KUKA KRL program: MyProgram_332().src

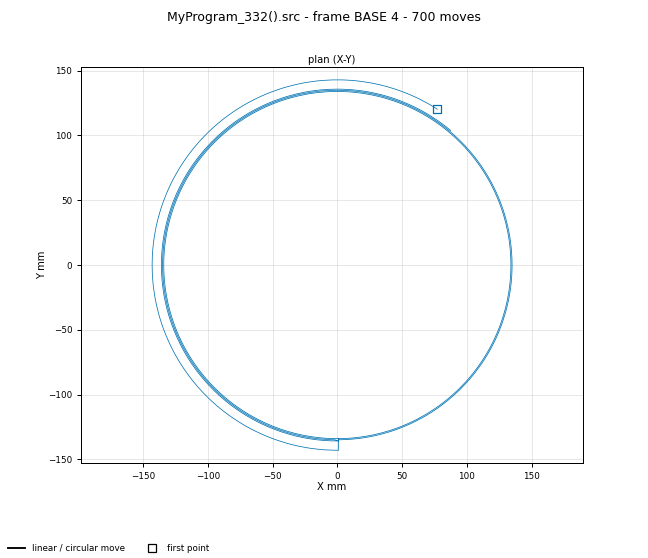
[picture p0: tool path of MyProgram_332().src in frame BASE 4, 700 of 700 moves have a stored position in this frame; points joined in program order, loops and branches not executed]
&ACCESS RVP
&REL 1
&PARAM TEMPLATE = C:\KRC\Roboter\Template\vorgabe
&PARAM EDITMASK = *
DEF MyProgram_332()
; ---- Setting reference (Base) ----
$BASE = BASE_DATA[4]

; --------------------------
; ---- Setting tool (TCP) ----
$TOOL = TOOL_DATA[3]
; --------------------------

$VEL.CP = VEL_APROX_PRINT
Startdeposition()
$VEL.CP = VEL_PRINT
LIN {X 77.191,Y 120.2651,Z 188,A 58.092,B 2.0692,C 0.0181,E1 2.1591,E2 395.982} C_DIS
LIN {X 74.024,Y 122.2399,Z 188,A 59.6872,B 2.0692,C 0.0151,E1 2.1552,E2 394.3743} C_DIS
LIN {X 70.243,Y 124.4513,Z 188,A 61.3886,B 2.0692,C 0.0127,E1 2.1511,E2 392.68} C_DIS
LIN {X 66.2155,Y 126.6377,Z 188,A 63.0311,B 2.0692,C 0.0112,E1 2.1471,E2 391.0624} C_DIS
LIN {X 63.4526,Y 128.0444,Z 188,A 64.253,B 2.0692,C 0.0096,E1 2.1441,E2 389.8433} C_DIS
LIN {X 60.2963,Y 129.5609,Z 188,A 65.6115,B 2.0692,C 0.008,E1 2.1406,E2 388.4907} C_DIS
LIN {X 55.8819,Y 131.5277,Z 188,A 67.6043,B 2.0692,C 0.0052,E1 2.1355,E2 386.4914} C_DIS
LIN {X 52.6403,Y 132.8581,Z 188,A 68.8611,B 2.0692,C 0.0043,E1 2.1323,E2 385.2535} C_DIS
LIN {X 48.7435,Y 134.3344,Z 188,A 70.5912,B 2.0692,C 0.0021,E1 2.1277,E2 383.5161} C_DIS
LIN {X 44.3687,Y 135.8443,Z 188,A 72.2898,B 2.0692,C 0.001,E1 2.1233,E2 381.8378} C_DIS
LIN {X 41.0274,Y 136.8906,Z 188,A 73.6584,B 2.0692,C -0.0002,E1 2.1196,E2 380.4739} C_DIS
LIN {X 37.6632,Y 137.8543,Z 188,A 75.0254,B 2.0692,C -0.0013,E1 2.116,E2 379.1118} C_DIS
LIN {X 34.5916,Y 138.6556,Z 188,A 76.3115,B 2.0692,C -0.0025,E1 2.1125,E2 377.8243} C_DIS
LIN {X 30.8569,Y 139.5349,Z 188,A 77.7931,B 2.0692,C -0.0035,E1 2.1084,E2 376.3503} C_DIS
LIN {X 27.4281,Y 140.2487,Z 188,A 79.1749,B 2.0692,C -0.0044,E1 2.1047,E2 374.9717} C_DIS
LIN {X 23.9731,Y 140.8799,Z 188,A 80.548,B 2.0692,C -0.0052,E1 2.1009,E2 373.6034} C_DIS
LIN {X 20.5127,Y 141.4248,Z 188,A 81.9382,B 2.0692,C -0.0059,E1 2.097,E2 372.2154} C_DIS
LIN {X 17.0406,Y 141.8848,Z 188,A 83.3239,B 2.0692,C -0.0066,E1 2.0932,E2 370.8325} C_DIS
LIN {X 13.9922,Y 142.2182,Z 188,A 84.541,B 2.0692,C -0.0072,E1 2.0898,E2 369.6174} C_DIS
LIN {X 10.0484,Y 142.5512,Z 188,A 86.0421,B 2.0692,C -0.0074,E1 2.0856,E2 368.1276} C_DIS
LIN {X 6.5517,Y 142.7556,Z 188,A 87.4775,B 2.0692,C -0.008,E1 2.0816,E2 366.6888} C_DIS
LIN {X 3.0497,Y 142.8736,Z 188,A 88.8217,B 2.0692,C -0.0081,E1 2.0779,E2 365.3528} C_DIS
LIN {X -0.4713,Y 142.9042,Z 188,A 90.1816,B 2.0692,C -0.0081,E1 2.0741,E2 363.9999} C_DIS
LIN {X -3.5202,Y 142.8619,Z 188,A 91.5285,B 2.0692,C -0.0089,E1 2.0703,E2 362.638} C_DIS
LIN {X -7.0204,Y 142.732,Z 188,A 92.9209,B 2.0692,C -0.009,E1 2.0664,E2 361.2477} C_DIS
LIN {X -10.515,Y 142.5171,Z 188,A 94.3659,B 2.0692,C -0.0092,E1 2.0623,E2 359.7981} C_DIS
LIN {X -14.0178,Y 142.2157,Z 188,A 95.7243,B 2.0692,C -0.0089,E1 2.0586,E2 358.4468} C_DIS
LIN {X -17.742,Y 141.8011,Z 188,A 97.2221,B 2.0692,C -0.0087,E1 2.0544,E2 356.9504} C_DIS
LIN {X -21.4322,Y 141.2887,Z 188,A 98.5946,B 2.0692,C -0.0079,E1 2.0506,E2 355.5936} C_DIS
LIN {X -24.4377,Y 140.8013,Z 188,A 99.9804,B 2.0692,C -0.0082,E1 2.0468,E2 354.1879} C_DIS
LIN {X -28.0983,Y 140.1152,Z 188,A 101.4739,B 2.0692,C -0.0077,E1 2.0427,E2 352.695} C_DIS
LIN {X -31.615,Y 139.3634,Z 188,A 102.9621,B 2.0692,C -0.0073,E1 2.0386,E2 351.2019} C_DIS
LIN {X -35.1507,Y 138.5137,Z 188,A 104.3003,B 2.0692,C -0.0061,E1 2.035,E2 349.8794} C_DIS
LIN {X -38.0927,Y 137.7342,Z 188,A 105.6465,B 2.0692,C -0.006,E1 2.0313,E2 348.5182} C_DIS
LIN {X -41.5005,Y 136.7458,Z 188,A 107.0908,B 2.0692,C -0.0052,E1 2.0274,E2 347.0718} C_DIS
LIN {X -44.8396,Y 135.6875,Z 188,A 108.5183,B 2.0692,C -0.0043,E1 2.0236,E2 345.6422} C_DIS
LIN {X -48.5796,Y 134.3935,Z 188,A 110.0373,B 2.0692,C -0.0029,E1 2.0196,E2 344.1326} C_DIS
LIN {X -51.4333,Y 133.3279,Z 188,A 111.38,B 2.0692,C -0.0023,E1 2.0161,E2 342.7755} C_DIS
LIN {X -54.7039,Y 132.0197,Z 188,A 112.8223,B 2.0692,C -0.0012,E1 2.0123,E2 341.3303} C_DIS
LIN {X -58.5883,Y 130.342,Z 188,A 114.6032,B 2.0692,C 0.0002,E1 2.0077,E2 339.5398} C_DIS
LIN {X -62.7858,Y 128.3734,Z 188,A 116.4246,B 2.0692,C 0.0022,E1 2.0031,E2 337.7243} C_DIS
LIN {X -66.0001,Y 126.7508,Z 188,A 118.0003,B 2.0692,C 0.0034,E1 1.9992,E2 336.1329} C_DIS
LIN {X -69.6929,Y 124.7605,Z 188,A 119.815,B 2.0692,C 0.005,E1 1.9947,E2 334.3027} C_DIS
LIN {X -73.4806,Y 122.5678,Z 188,A 121.54,B 2.0692,C 0.0073,E1 1.9905,E2 332.5826} C_DIS
LIN {X -77.1982,Y 120.2605,Z 188,A 123.3495,B 2.0692,C 0.0095,E1 1.9862,E2 330.7672} C_DIS
LIN {X -80.8424,Y 117.8416,Z 188,A 125.2463,B 2.0692,C 0.0116,E1 1.9818,E2 328.8536} C_DIS
LIN {X -84.6161,Y 115.1618,Z 188,A 127.1705,B 2.0692,C 0.0142,E1 1.9774,E2 326.9219} C_DIS
LIN {X -88.4338,Y 112.257,Z 188,A 129.1398,B 2.0692,C 0.0171,E1 1.9731,E2 324.9481} C_DIS
LIN {X -92.0062,Y 109.3481,Z 188,A 131.0239,B 2.0692,C 0.0201,E1 1.969,E2 323.0606} C_DIS
LIN {X -95.3272,Y 106.4653,Z 188,A 132.9387,B 2.0692,C 0.0228,E1 1.9649,E2 321.1277} C_DIS
LIN {X -98.5443,Y 103.4949,Z 188,A 134.7156,B 2.0692,C 0.0259,E1 1.9613,E2 319.3494} C_DIS
LIN {X -101.669,Y 100.4276,Z 188,A 136.5545,B 2.0691,C 0.029,E1 1.9576,E2 317.5011} C_DIS
LIN {X -104.6976,Y 97.2654,Z 188,A 138.3926,B 2.0691,C 0.0322,E1 1.9541,E2 315.6537} C_DIS
LIN {X -107.4912,Y 94.1692,Z 188,A 140.2044,B 2.069,C 0.0352,E1 1.9507,E2 313.8253} C_DIS
LIN {X -110.3256,Y 90.8325,Z 188,A 142.0599,B 2.069,C 0.0386,E1 1.9474,E2 311.9582} C_DIS
LIN {X -113.1958,Y 87.2296,Z 188,A 143.9226,B 2.0689,C 0.0425,E1 1.9441,E2 310.0948} C_DIS
LIN {X -115.4534,Y 84.219,Z 188,A 145.6429,B 2.0689,C 0.0454,E1 1.9412,E2 308.3484} C_DIS
LIN {X -117.9768,Y 80.6453,Z 188,A 147.4532,B 2.0687,C 0.0492,E1 1.9383,E2 306.5321} C_DIS
LIN {X -120.265,Y 77.1912,Z 188,A 149.2357,B 2.0687,C 0.0527,E1 1.9356,E2 304.7352} C_DIS
LIN {X -122.6861,Y 73.282,Z 188,A 151.1891,B 2.0685,C 0.0568,E1 1.9328,E2 302.7689} C_DIS
LIN {X -125.0733,Y 69.1289,Z 188,A 153.1628,B 2.0684,C 0.0613,E1 1.93,E2 300.7897} C_DIS
LIN {X -127.0339,Y 65.4554,Z 188,A 154.8401,B 2.0683,C 0.0654,E1 1.9279,E2 299.1126} C_DIS
LIN {X -128.5394,Y 62.4493,Z 188,A 156.4673,B 2.0682,C 0.0682,E1 1.9258,E2 297.4501} C_DIS
LIN {X -130.2908,Y 58.7026,Z 188,A 158.1973,B 2.068,C 0.0723,E1 1.9238,E2 295.7119} C_DIS
LIN {X -132.0308,Y 54.6774,Z 188,A 160.0188,B 2.0679,C 0.0766,E1 1.9218,E2 293.8834} C_DIS
LIN {X -133.4949,Y 51.0035,Z 188,A 161.6693,B 2.0677,C 0.0806,E1 1.9201,E2 292.2255} C_DIS
LIN {X -134.5486,Y 48.1494,Z 188,A 163.0215,B 2.0677,C 0.0836,E1 1.9188,E2 290.8568} C_DIS
LIN {X -135.8334,Y 44.4014,Z 188,A 164.6773,B 2.0674,C 0.0877,E1 1.9173,E2 289.1933} C_DIS
LIN {X -136.8857,Y 41.0433,Z 188,A 166.1859,B 2.0673,C 0.0913,E1 1.9161,E2 287.673} C_DIS
LIN {X -137.8633,Y 37.6301,Z 188,A 167.6986,B 2.0671,C 0.0949,E1 1.9149,E2 286.1495} C_DIS
LIN {X -138.639,Y 34.6571,Z 188,A 169.091,B 2.067,C 0.098,E1 1.914,E2 284.7367} C_DIS
LIN {X -139.5401,Y 30.8326,Z 188,A 170.7279,B 2.0668,C 0.1022,E1 1.9129,E2 283.0928} C_DIS
LIN {X -140.2508,Y 27.417,Z 188,A 172.2387,B 2.0666,C 0.1058,E1 1.9121,E2 281.568} C_DIS
LIN {X -140.8821,Y 23.9599,Z 188,A 173.5765,B 2.0664,C 0.1098,E1 1.9115,E2 280.2406} C_DIS
LIN {X -141.4257,Y 20.5062,Z 188,A 175.2435,B 2.0662,C 0.1133,E1 1.9107,E2 278.5393} C_DIS
LIN {X -141.8873,Y 17.0199,Z 188,A 176.7542,B 2.066,C 0.117,E1 1.9102,E2 277.0161} C_DIS
LIN {X -142.218,Y 13.9942,Z 188,A 178.0706,B 2.0658,C 0.1203,E1 1.9098,E2 275.6878} C_DIS
LIN {X -142.5505,Y 10.0574,Z 188,A 179.869,B 2.0656,C 0.1244,E1 1.9094,E2 273.8617} C_DIS
LIN {X -142.7564,Y 6.5367,Z 188,A -178.7374,B 2.0653,C 0.1284,E1 1.9092,E2 272.4718} C_DIS
LIN {X -142.8738,Y 3.0367,Z 188,A -177.1408,B 2.0651,C 0.132,E1 1.9092,E2 270.8502} C_DIS
LIN {X -142.9079,Y -0.008,Z 188,A -175.833,B 2.0649,C 0.1353,E1 1.9092,E2 269.5315} C_DIS
LIN {X -142.8622,Y -3.5089,Z 188,A -174.3736,B 2.0646,C 0.1391,E1 1.9092,E2 268.0654} C_DIS
LIN {X -142.7304,Y -7.0533,Z 188,A -172.8568,B 2.0644,C 0.1429,E1 1.9094,E2 266.5366} C_DIS
LIN {X -142.515,Y -10.5447,Z 188,A -171.3087,B 2.0641,C 0.1466,E1 1.9097,E2 264.9696} C_DIS
LIN {X -142.2149,Y -14.026,Z 188,A -169.8577,B 2.0638,C 0.1504,E1 1.9101,E2 263.5126} C_DIS
LIN {X -141.829,Y -17.5087,Z 188,A -168.3528,B 2.0636,C 0.1541,E1 1.9106,E2 261.9949} C_DIS
LIN {X -141.2849,Y -21.4566,Z 188,A -166.7811,B 2.0632,C 0.1586,E1 1.9112,E2 260.4277} C_DIS
LIN {X -140.7997,Y -24.4466,Z 188,A -165.3118,B 2.063,C 0.1615,E1 1.9119,E2 258.9244} C_DIS
LIN {X -140.1632,Y -27.8624,Z 188,A -163.7546,B 2.0627,C 0.165,E1 1.9127,E2 257.3455} C_DIS
LIN {X -139.4338,Y -31.307,Z 188,A -162.2535,B 2.0624,C 0.1687,E1 1.9136,E2 255.8329} C_DIS
LIN {X -138.5086,Y -35.1708,Z 188,A -160.7176,B 2.062,C 0.1731,E1 1.9146,E2 254.3056} C_DIS
LIN {X -137.7274,Y -38.1169,Z 188,A -159.2967,B 2.0618,C 0.176,E1 1.9157,E2 252.8579} C_DIS
LIN {X -136.7515,Y -41.482,Z 188,A -157.7941,B 2.0615,C 0.1796,E1 1.9169,E2 251.3426} C_DIS
LIN {X -135.6907,Y -44.8301,Z 188,A -156.2473,B 2.0612,C 0.183,E1 1.9182,E2 249.7774} C_DIS
LIN {X -134.3907,Y -48.5874,Z 188,A -154.503,B 2.0608,C 0.1869,E1 1.9199,E2 248.013} C_DIS
LIN {X -132.6867,Y -53.0655,Z 188,A -152.4738,B 2.0604,C 0.1916,E1 1.922,E2 245.9696} C_DIS
LIN {X -131.3491,Y -56.2955,Z 188,A -150.9828,B 2.0601,C 0.1949,E1 1.9236,E2 244.4668} C_DIS
LIN {X -129.9323,Y -59.4931,Z 188,A -149.5427,B 2.0598,C 0.1984,E1 1.9253,E2 243.0219} C_DIS
LIN {X -128.426,Y -62.6791,Z 188,A -148.0459,B 2.0594,C 0.2017,E1 1.9271,E2 241.5141} C_DIS
LIN {X -126.7358,Y -66.0287,Z 188,A -146.4049,B 2.0591,C 0.205,E1 1.9292,E2 239.8545} C_DIS
LIN {X -124.7679,Y -69.6797,Z 188,A -144.5415,B 2.0588,C 0.2086,E1 1.9317,E2 237.9637} C_DIS
LIN {X -122.575,Y -73.4685,Z 188,A -142.7546,B 2.0584,C 0.2126,E1 1.9343,E2 236.1729} C_DIS
LIN {X -120.2459,Y -77.221,Z 188,A -140.9018,B 2.058,C 0.2165,E1 1.9371,E2 234.3091} C_DIS
LIN {X -117.8382,Y -80.8473,Z 188,A -138.9752,B 2.0576,C 0.2199,E1 1.9401,E2 232.3575} C_DIS
LIN {X -115.1519,Y -84.6296,Z 188,A -137.0086,B 2.0572,C 0.2237,E1 1.9434,E2 230.3764} C_DIS
LIN {X -112.2516,Y -88.4406,Z 188,A -135.0163,B 2.0568,C 0.2276,E1 1.9468,E2 228.3743} C_DIS
LIN {X -109.3488,Y -92.0054,Z 188,A -133.1154,B 2.0563,C 0.2312,E1 1.9502,E2 226.4656} C_DIS
LIN {X -106.4681,Y -95.324,Z 188,A -131.193,B 2.056,C 0.2342,E1 1.9538,E2 224.5208} C_DIS
LIN {X -103.4984,Y -98.5407,Z 188,A -129.4109,B 2.0556,C 0.2375,E1 1.9572,E2 222.7351} C_DIS
LIN {X -100.4313,Y -101.6653,Z 188,A -127.5694,B 2.0553,C 0.2405,E1 1.9609,E2 220.8816} C_DIS
LIN {X -97.2556,Y -104.7068,Z 188,A -125.7391,B 2.0549,C 0.2435,E1 1.9646,E2 219.042} C_DIS
LIN {X -94.1794,Y -107.4823,Z 188,A -123.9498,B 2.0546,C 0.2459,E1 1.9684,E2 217.2346} C_DIS
LIN {X -90.8327,Y -110.3255,Z 188,A -122.1095,B 2.0543,C 0.2486,E1 1.9724,E2 215.3829} C_DIS
LIN {X -87.2268,Y -113.1979,Z 188,A -120.1487,B 2.054,C 0.2511,E1 1.9767,E2 213.4062} C_DIS
LIN {X -83.5252,Y -115.9562,Z 188,A -118.2289,B 2.0537,C 0.2536,E1 1.9811,E2 211.4764} C_DIS
LIN {X -80.1185,Y -118.3349,Z 188,A -116.5271,B 2.0534,C 0.2558,E1 1.985,E2 209.7695} C_DIS
LIN {X -76.4552,Y -120.7343,Z 188,A -114.7741,B 2.0531,C 0.2582,E1 1.9891,E2 208.0167} C_DIS
LIN {X -72.7203,Y -123.0205,Z 188,A -112.9568,B 2.0529,C 0.2602,E1 1.9935,E2 206.1906} C_DIS
LIN {X -68.8933,Y -125.2038,Z 188,A -111.1836,B 2.0526,C 0.2622,E1 1.9979,E2 204.4161} C_DIS
LIN {X -65.6011,Y -126.9597,Z 188,A -109.6543,B 2.0524,C 0.2638,E1 2.0017,E2 202.8819} C_DIS
LIN {X -62.4691,Y -128.5296,Z 188,A -108.2013,B 2.0523,C 0.265,E1 2.0053,E2 201.4217} C_DIS
LIN {X -58.7094,Y -130.2878,Z 188,A -106.4164,B 2.0521,C 0.2662,E1 2.0099,E2 199.6191} C_DIS
LIN {X -54.6923,Y -132.0246,Z 188,A -104.6725,B 2.0519,C 0.2678,E1 2.0144,E2 197.8764} C_DIS
LIN {X -51.0039,Y -133.4948,Z 188,A -102.9249,B 2.0519,C 0.2684,E1 2.019,E2 196.1061} C_DIS
LIN {X -46.0363,Y -135.2883,Z 188,A -100.9306,B 2.0516,C 0.2704,E1 2.0242,E2 194.129} C_DIS
LIN {X -42.7082,Y -136.3755,Z 188,A -99.5065,B 2.0515,C 0.2712,E1 2.0281,E2 192.7017} C_DIS
LIN {X -39.3559,Y -137.3805,Z 188,A -98.0852,B 2.0514,C 0.2719,E1 2.0319,E2 191.2773} C_DIS
LIN {X -36.4217,Y -138.1855,Z 188,A -96.8427,B 2.0513,C 0.2724,E1 2.0353,E2 190.0311} C_DIS
LIN {X -32.5698,Y -139.1453,Z 188,A -95.2317,B 2.0513,C 0.273,E1 2.0396,E2 188.417} C_DIS
LIN {X -29.1419,Y -139.9029,Z 188,A -93.8108,B 2.0512,C 0.2735,E1 2.0435,E2 186.9936} C_DIS
LIN {X -25.7011,Y -140.5752,Z 188,A -92.3963,B 2.0512,C 0.2739,E1 2.0474,E2 185.5772} C_DIS
LIN {X -22.7005,Y -141.0922,Z 188,A -91.0483,B 2.0512,C 0.2735,E1 2.0512,E2 184.2106} C_DIS
LIN {X -18.7821,Y -141.6649,Z 188,A -89.5751,B 2.051,C 0.2743,E1 2.0553,E2 182.7531} C_DIS
LIN {X -15.2873,Y -142.0844,Z 188,A -88.2632,B 2.051,C 0.2749,E1 2.0589,E2 181.455} C_DIS
LIN {X -12.2533,Y -142.3783,Z 188,A -86.8704,B 2.051,C 0.2741,E1 2.0628,E2 180.037} C_DIS
LIN {X -8.7592,Y -142.6358,Z 188,A -85.4919,B 2.051,C 0.2741,E1 2.0667,E2 178.6617} C_DIS
LIN {X -4.8038,Y -142.8258,Z 188,A -83.9134,B 2.051,C 0.2741,E1 2.0711,E2 177.0838} C_DIS
LIN {X -1.7417,Y -142.8954,Z 188,A -82.6323,B 2.0512,C 0.2735,E1 2.0747,E2 175.7945} C_DIS
LIN {X 1.0451,Y -142.9001,Z 188,A -81.9408,B 2.0509,C 0.2755,E1 2.0765,E2 175.1638} C_DIS
Enddeposition()
LIN {X 0.9696,Y -133.9381,Z 189,A -81.2734,B 1.7006,C 0.247,E1 1.727,E2 174.2111} C_DIS
Startdeposition()
$VEL.CP = VEL_PRINT
LIN {X -1.6562,Y -133.9352,Z 189,A -82.7535,B 1.7004,C 0.2488,E1 1.7227,E2 175.7398} C_DIS
LIN {X -4.9327,Y -133.8536,Z 189,A -84.2094,B 1.7003,C 0.2493,E1 1.7186,E2 177.2035} C_DIS
LIN {X -8.9898,Y -133.6442,Z 189,A -85.8795,B 1.7003,C 0.2492,E1 1.714,E2 178.8655} C_DIS
LIN {X -12.2534,Y -133.3835,Z 189,A -87.2736,B 1.7003,C 0.2492,E1 1.7101,E2 180.2593} C_DIS
LIN {X -15.6691,Y -133.0245,Z 189,A -88.7363,B 1.7003,C 0.2492,E1 1.706,E2 181.7218} C_DIS
LIN {X -18.9216,Y -132.6008,Z 189,A -90.1407,B 1.7003,C 0.249,E1 1.7021,E2 183.1269} C_DIS
LIN {X -22.1631,Y -132.0976,Z 189,A -91.551,B 1.7003,C 0.2488,E1 1.6982,E2 184.5387} C_DIS
LIN {X -25.4054,Y -131.5127,Z 189,A -92.9674,B 1.7004,C 0.2484,E1 1.6943,E2 185.9566} C_DIS
LIN {X -28.6288,Y -130.8491,Z 189,A -94.3882,B 1.7004,C 0.248,E1 1.6904,E2 187.3796} C_DIS
LIN {X -31.8278,Y -130.1082,Z 189,A -95.8093,B 1.7005,C 0.2476,E1 1.6865,E2 188.8034} C_DIS
LIN {X -35.0075,Y -129.2891,Z 189,A -97.2218,B 1.7006,C 0.247,E1 1.6827,E2 190.2175} C_DIS
LIN {X -38.1643,Y -128.3928,Z 189,A -98.6609,B 1.7007,C 0.2464,E1 1.6788,E2 191.6617} C_DIS
LIN {X -41.8745,Y -127.2307,Z 189,A -100.4022,B 1.7008,C 0.2456,E1 1.6741,E2 193.4139} C_DIS
LIN {X -45.1417,Y -126.108,Z 189,A -101.8618,B 1.701,C 0.2446,E1 1.6702,E2 194.8714} C_DIS
LIN {X -48.912,Y -124.6944,Z 189,A -103.6411,B 1.7011,C 0.2435,E1 1.6656,E2 196.6588} C_DIS
LIN {X -51.948,Y -123.4602,Z 189,A -105.064,B 1.7013,C 0.2424,E1 1.6619,E2 198.0848} C_DIS
LIN {X -54.9538,Y -122.1518,Z 189,A -106.5236,B 1.7014,C 0.2413,E1 1.6581,E2 199.5522} C_DIS
LIN {X -58.7511,Y -120.3724,Z 189,A -108.3429,B 1.7017,C 0.2396,E1 1.6535,E2 201.3753} C_DIS
LIN {X -61.6882,Y -118.8944,Z 189,A -109.7765,B 1.7019,C 0.2383,E1 1.6499,E2 202.8127} C_DIS
LIN {X -65.265,Y -116.9704,Z 189,A -111.6349,B 1.7021,C 0.2367,E1 1.6453,E2 204.6874} C_DIS
LIN {X -68.2395,Y -115.2603,Z 189,A -113.1191,B 1.7023,C 0.235,E1 1.6417,E2 206.1741} C_DIS
LIN {X -71.6626,Y -113.1633,Z 189,A -114.9315,B 1.7026,C 0.233,E1 1.6374,E2 207.9992} C_DIS
LIN {X -75.1549,Y -110.8746,Z 189,A -116.7644,B 1.7029,C 0.2307,E1 1.6331,E2 209.8385} C_DIS
LIN {X -77.7315,Y -109.0838,Z 189,A -118.1997,B 1.7031,C 0.2291,E1 1.6297,E2 211.2861} C_DIS
LIN {X -80.513,Y -107.0473,Z 189,A -119.6835,B 1.7034,C 0.2269,E1 1.6264,E2 212.7711} C_DIS
LIN {X -83.3511,Y -104.8524,Z 189,A -121.3995,B 1.7037,C 0.225,E1 1.6226,E2 214.5111} C_DIS
LIN {X -86.5851,Y -102.1983,Z 189,A -123.2754,B 1.704,C 0.2223,E1 1.6185,E2 216.3983} C_DIS
LIN {X -89.7072,Y -99.4696,Z 189,A -125.1588,B 1.7044,C 0.2195,E1 1.6145,E2 218.2961} C_DIS
LIN {X -92.719,Y -96.6678,Z 189,A -126.9845,B 1.7048,C 0.2165,E1 1.6108,E2 220.1303} C_DIS
LIN {X -95.5597,Y -93.8604,Z 189,A -128.8114,B 1.7051,C 0.2136,E1 1.6072,E2 221.9726} C_DIS
LIN {X -98.393,Y -90.8864,Z 189,A -130.6917,B 1.7055,C 0.2105,E1 1.6035,E2 223.8688} C_DIS
LIN {X -101.1837,Y -87.7692,Z 189,A -132.5791,B 1.7059,C 0.2072,E1 1.6,E2 225.7687} C_DIS
LIN {X -103.7757,Y -84.6879,Z 189,A -134.4013,B 1.7063,C 0.2038,E1 1.5967,E2 227.6035} C_DIS
LIN {X -106.3702,Y -81.4052,Z 189,A -136.3037,B 1.7067,C 0.2003,E1 1.5934,E2 229.5203} C_DIS
LIN {X -108.5512,Y -78.4735,Z 189,A -137.9487,B 1.7071,C 0.197,E1 1.5907,E2 231.1756} C_DIS
LIN {X -110.9952,Y -74.9767,Z 189,A -139.9984,B 1.7075,C 0.1933,E1 1.5874,E2 233.2539} C_DIS
LIN {X -113.1673,Y -71.6563,Z 189,A -141.6742,B 1.708,C 0.1895,E1 1.5849,E2 234.9265} C_DIS
LIN {X -114.8894,Y -68.8619,Z 189,A -143.3374,B 1.7083,C 0.1866,E1 1.5824,E2 236.6228} C_DIS
LIN {X -116.9818,Y -65.2446,Z 189,A -145.112,B 1.7088,C 0.1823,E1 1.58,E2 238.3953} C_DIS
LIN {X -118.8071,Y -61.8544,Z 189,A -146.9061,B 1.7092,C 0.1786,E1 1.5776,E2 240.2077} C_DIS
LIN {X -120.372,Y -58.7518,Z 189,A -148.4868,B 1.7095,C 0.175,E1 1.5756,E2 241.8} C_DIS
LIN {X -121.999,Y -55.2954,Z 189,A -150.3655,B 1.7099,C 0.1712,E1 1.5734,E2 243.7094} C_DIS
LIN {X -123.7488,Y -51.257,Z 189,A -152.2921,B 1.7104,C 0.1665,E1 1.5712,E2 245.6409} C_DIS
LIN {X -124.9682,Y -48.2075,Z 189,A -153.8327,B 1.7107,C 0.1631,E1 1.5697,E2 247.1983} C_DIS
LIN {X -126.4045,Y -44.3061,Z 189,A -155.9166,B 1.7111,C 0.1587,E1 1.5677,E2 249.3201} C_DIS
LIN {X -127.9219,Y -39.7142,Z 189,A -158.0785,B 1.7116,C 0.1533,E1 1.5658,E2 251.493} C_DIS
LIN {X -129.0888,Y -35.7373,Z 189,A -159.9092,B 1.712,C 0.1487,E1 1.5644,E2 253.3301} C_DIS
LIN {X -129.9304,Y -32.5454,Z 189,A -161.4449,B 1.7123,C 0.145,E1 1.5633,E2 254.8808} C_DIS
LIN {X -130.6896,Y -29.3499,Z 189,A -162.9723,B 1.7126,C 0.1412,E1 1.5623,E2 256.423} C_DIS
LIN {X -131.3708,Y -26.1344,Z 189,A -164.5006,B 1.7129,C 0.1375,E1 1.5615,E2 257.9659} C_DIS
LIN {X -131.9747,Y -22.8945,Z 189,A -166.0329,B 1.7132,C 0.1337,E1 1.5607,E2 259.5129} C_DIS
LIN {X -132.4964,Y -19.6519,Z 189,A -167.5916,B 1.7135,C 0.1299,E1 1.56,E2 261.0901} C_DIS
LIN {X -132.9006,Y -16.7013,Z 189,A -169.0642,B 1.7138,C 0.1265,E1 1.5595,E2 262.5868} C_DIS
LIN {X -133.2991,Y -13.1322,Z 189,A -170.6537,B 1.7141,C 0.1223,E1 1.559,E2 264.182} C_DIS
LIN {X -133.5815,Y -9.8488,Z 189,A -172.1826,B 1.7144,C 0.1184,E1 1.5587,E2 265.725} C_DIS
LIN {X -133.7949,Y -6.3332,Z 189,A -173.9256,B 1.7146,C 0.1144,E1 1.5584,E2 267.4964} C_DIS
LIN {X -133.923,Y -2.3881,Z 189,A -175.6855,B 1.715,C 0.1097,E1 1.5583,E2 269.264} C_DIS
LIN {X -133.9355,Y 1.6379,Z 189,A -177.5708,B 1.7152,C 0.1049,E1 1.5583,E2 271.1685} C_DIS
LIN {X -133.8537,Y 4.9287,Z 189,A -179.24,B 1.7155,C 0.1011,E1 1.5584,E2 272.8688} C_DIS
LIN {X -133.6462,Y 8.9572,Z 189,A 179.02,B 1.7158,C 0.0963,E1 1.5587,E2 274.6096} C_DIS
LIN {X -133.3858,Y 12.2294,Z 189,A 177.481,B 1.716,C 0.0925,E1 1.5591,E2 276.1642} C_DIS
LIN {X -133.0265,Y 15.6524,Z 189,A 175.8452,B 1.7162,C 0.0885,E1 1.5596,E2 277.819} C_DIS
LIN {X -132.4956,Y 19.6574,Z 189,A 174.0125,B 1.7164,C 0.0837,E1 1.5603,E2 279.6633} C_DIS
LIN {X -132.029,Y 22.5747,Z 189,A 172.568,B 1.7166,C 0.0803,E1 1.561,E2 281.1289} C_DIS
LIN {X -131.3718,Y 26.1298,Z 189,A 170.7691,B 1.7168,C 0.0762,E1 1.562,E2 282.9572} C_DIS
LIN {X -130.5677,Y 29.8837,Z 189,A 169.0808,B 1.717,C 0.0718,E1 1.563,E2 284.6499} C_DIS
LIN {X -129.5151,Y 34.1601,Z 189,A 167.082,B 1.7172,C 0.0668,E1 1.5644,E2 286.6613} C_DIS
LIN {X -128.3868,Y 38.1848,Z 189,A 165.1561,B 1.7173,C 0.0621,E1 1.5659,E2 288.6026} C_DIS
LIN {X -127.4124,Y 41.3202,Z 189,A 163.6391,B 1.7175,C 0.0584,E1 1.5672,E2 290.1321} C_DIS
LIN {X -126.3617,Y 44.4295,Z 189,A 162.1029,B 1.7175,C 0.0548,E1 1.5686,E2 291.6831} C_DIS
LIN {X -125.2905,Y 47.3642,Z 189,A 160.6527,B 1.7177,C 0.0514,E1 1.57,E2 293.1459} C_DIS
LIN {X -124.0329,Y 50.5669,Z 189,A 158.8948,B 1.7177,C 0.0478,E1 1.5719,E2 294.9367} C_DIS
LIN {X -122.4561,Y 54.2733,Z 189,A 157.2487,B 1.7179,C 0.0434,E1 1.5737,E2 296.5725} C_DIS
LIN {X -121.391,Y 56.6155,Z 189,A 155.8582,B 1.7179,C 0.0409,E1 1.5753,E2 297.9966} C_DIS
LIN {X -119.638,Y 60.2327,Z 189,A 154.1549,B 1.7181,C 0.0366,E1 1.5774,E2 299.6967} C_DIS
LIN {X -118.1271,Y 63.1467,Z 189,A 152.6371,B 1.7181,C 0.0333,E1 1.5794,E2 301.227} C_DIS
LIN {X -116.5454,Y 66.021,Z 189,A 150.99,B 1.7181,C 0.0302,E1 1.5817,E2 302.9016} C_DIS
LIN {X -114.4229,Y 69.6345,Z 189,A 149.1856,B 1.7183,C 0.026,E1 1.5843,E2 304.7062} C_DIS
LIN {X -112.6816,Y 72.4178,Z 189,A 147.6792,B 1.7183,C 0.0229,E1 1.5866,E2 306.2235} C_DIS
LIN {X -110.4528,Y 75.7734,Z 189,A 145.7927,B 1.7183,C 0.0191,E1 1.5896,E2 308.1279} C_DIS
LIN {X -108.0209,Y 79.2018,Z 189,A 143.9138,B 1.7183,C 0.0153,E1 1.5926,E2 310.0149} C_DIS
LIN {X -106.0981,Y 81.7603,Z 189,A 142.3569,B 1.7184,C 0.0126,E1 1.5953,E2 311.5926} C_DIS
LIN {X -103.5442,Y 84.9712,Z 189,A 140.4601,B 1.7184,C 0.0091,E1 1.5987,E2 313.5046} C_DIS
LIN {X -100.63,Y 88.4036,Z 189,A 138.4163,B 1.7184,C 0.0054,E1 1.6024,E2 315.5607} C_DIS
LIN {X -97.8243,Y 91.4982,Z 189,A 136.5504,B 1.7184,C 0.002,E1 1.606,E2 317.4345} C_DIS
LIN {X -94.9779,Y 94.449,Z 189,A 134.7023,B 1.7184,C -0.0012,E1 1.6096,E2 319.2921} C_DIS
LIN {X -92.0796,Y 97.277,Z 189,A 132.8399,B 1.7184,C -0.0041,E1 1.6134,E2 321.1683} C_DIS
LIN {X -89.0574,Y 100.0518,Z 189,A 130.9759,B 1.7184,C -0.007,E1 1.6173,E2 323.0436} C_DIS
LIN {X -85.9529,Y 102.7305,Z 189,A 129.1513,B 1.7184,C -0.0098,E1 1.6212,E2 324.8751} C_DIS
LIN {X -82.7673,Y 105.3138,Z 189,A 127.312,B 1.7184,C -0.0125,E1 1.6252,E2 326.7228} C_DIS
LIN {X -79.1869,Y 108.0318,Z 189,A 125.3488,B 1.7184,C -0.0153,E1 1.6297,E2 328.6893} C_DIS
LIN {X -75.7755,Y 110.4514,Z 189,A 123.5087,B 1.7184,C -0.0178,E1 1.6339,E2 330.5341} C_DIS
LIN {X -73.0462,Y 112.2751,Z 189,A 122.0421,B 1.7184,C -0.0196,E1 1.6373,E2 332.007} C_DIS
LIN {X -70.2594,Y 114.0399,Z 189,A 120.5811,B 1.7184,C -0.0213,E1 1.6408,E2 333.4727} C_DIS
LIN {X -66.8106,Y 116.0943,Z 189,A 118.7683,B 1.7183,C -0.0232,E1 1.6452,E2 335.2952} C_DIS
LIN {X -63.8176,Y 117.7662,Z 189,A 117.0997,B 1.7183,C -0.0245,E1 1.6494,E2 336.9858} C_DIS
LIN {X -60.5474,Y 119.4778,Z 189,A 115.5923,B 1.7183,C -0.0264,E1 1.6531,E2 338.4841} C_DIS
LIN {X -56.5809,Y 121.407,Z 189,A 113.6559,B 1.7183,C -0.0281,E1 1.658,E2 340.425} C_DIS
LIN {X -53.4468,Y 122.8187,Z 189,A 112.1862,B 1.7182,C -0.0295,E1 1.6618,E2 341.8937} C_DIS
LIN {X -49.8945,Y 124.304,Z 189,A 110.4685,B 1.7182,C -0.0307,E1 1.6663,E2 343.6185} C_DIS
LIN {X -45.9814,Y 125.8053,Z 189,A 108.6602,B 1.7182,C -0.032,E1 1.671,E2 345.4275} C_DIS
LIN {X -42.7433,Y 126.9414,Z 189,A 107.2026,B 1.7182,C -0.0331,E1 1.6749,E2 346.8831} C_DIS
LIN {X -39.7443,Y 127.9126,Z 189,A 105.6478,B 1.7182,C -0.0333,E1 1.6791,E2 348.4603} C_DIS
LIN {X -35.7151,Y 129.0949,Z 189,A 103.9618,B 1.7182,C -0.0346,E1 1.6836,E2 350.133} C_DIS
LIN {X -32.5393,Y 129.932,Z 189,A 102.5385,B 1.7181,C -0.0352,E1 1.6875,E2 351.5576} C_DIS
LIN {X -29.3438,Y 130.691,Z 189,A 101.1188,B 1.7181,C -0.0357,E1 1.6913,E2 352.9783} C_DIS
LIN {X -26.1308,Y 131.3716,Z 189,A 99.715,B 1.7181,C -0.0362,E1 1.6952,E2 354.3813} C_DIS
LIN {X -22.8752,Y 131.9782,Z 189,A 98.2755,B 1.7181,C -0.0365,E1 1.6992,E2 355.8227} C_DIS
LIN {X -19.6371,Y 132.4985,Z 189,A 96.8448,B 1.7181,C -0.0366,E1 1.7031,E2 357.2558} C_DIS
LIN {X -15.6659,Y 133.0249,Z 189,A 95.1237,B 1.7181,C -0.0368,E1 1.7079,E2 358.9769} C_DIS
LIN {X -12.2308,Y 133.3857,Z 189,A 93.6752,B 1.7181,C -0.0369,E1 1.712,E2 360.4215} C_DIS
LIN {X -8.9401,Y 133.6473,Z 189,A 92.2857,B 1.7181,C -0.0369,E1 1.7158,E2 361.8079} C_DIS
LIN {X -5.24,Y 133.8416,Z 189,A 90.6265,B 1.7181,C -0.0365,E1 1.7205,E2 363.4747} C_DIS
LIN {X -1.6342,Y 133.9355,Z 189,A 89.1182,B 1.7181,C -0.0363,E1 1.7247,E2 364.9785} C_DIS
LIN {X 2.3879,Y 133.923,Z 189,A 87.4179,B 1.7181,C -0.0359,E1 1.7295,E2 366.6759} C_DIS
LIN {X 5.6982,Y 133.8237,Z 189,A 86.0287,B 1.7181,C -0.0355,E1 1.7334,E2 368.0615} C_DIS
LIN {X 8.976,Y 133.6451,Z 189,A 84.6261,B 1.7181,C -0.035,E1 1.7373,E2 369.4634} C_DIS
LIN {X 12.2428,Y 133.3845,Z 189,A 83.2451,B 1.7181,C -0.0344,E1 1.7411,E2 370.8415} C_DIS
LIN {X 15.6618,Y 133.0254,Z 189,A 81.8067,B 1.7181,C -0.0337,E1 1.7451,E2 372.2758} C_DIS
LIN {X 18.9157,Y 132.6016,Z 189,A 80.4317,B 1.7181,C -0.0329,E1 1.749,E2 373.6471} C_DIS
LIN {X 22.1703,Y 132.0964,Z 189,A 79.0533,B 1.7181,C -0.0321,E1 1.7528,E2 375.0216} C_DIS
LIN {X 25.407,Y 131.5124,Z 189,A 77.6782,B 1.7181,C -0.0312,E1 1.7565,E2 376.3927} C_DIS
LIN {X 28.6253,Y 130.8499,Z 189,A 76.3064,B 1.7181,C -0.0302,E1 1.7603,E2 377.7603} C_DIS
LIN {X 31.8244,Y 130.109,Z 189,A 74.7915,B 1.7182,C -0.0285,E1 1.7644,E2 379.2873} C_DIS
LIN {X 36.1055,Y 128.9858,Z 189,A 73.0251,B 1.7182,C -0.0272,E1 1.7692,E2 381.0389} C_DIS
LIN {X 39.7914,Y 127.8982,Z 189,A 71.4996,B 1.7182,C -0.026,E1 1.7732,E2 382.5507} C_DIS
LIN {X 42.7506,Y 126.939,Z 189,A 70.1696,B 1.7182,C -0.0246,E1 1.7768,E2 383.8802} C_DIS
LIN {X 46.6769,Y 125.5479,Z 189,A 68.3549,B 1.7183,C -0.0224,E1 1.7816,E2 385.6983} C_DIS
LIN {X 50.5719,Y 124.0309,Z 189,A 66.6187,B 1.7183,C -0.0204,E1 1.7861,E2 387.4283} C_DIS
LIN {X 54.959,Y 122.1494,Z 189,A 64.7783,B 1.7183,C -0.0187,E1 1.7907,E2 389.2455} C_DIS
LIN {X 57.9375,Y 120.765,Z 189,A 63.3815,B 1.7183,C -0.0167,E1 1.7943,E2 390.6412} C_DIS
LIN {X 61.0641,Y 119.2148,Z 189,A 61.9242,B 1.7183,C -0.0147,E1 1.7979,E2 392.0943} C_DIS
LIN {X 65.2607,Y 116.9728,Z 189,A 60.0374,B 1.7184,C -0.0124,E1 1.8025,E2 393.964} C_DIS
LIN {X 68.8656,Y 114.8872,Z 189,A 58.3506,B 1.7184,C -0.0101,E1 1.8066,E2 395.6398} C_DIS
LIN {X 72.4087,Y 112.6875,Z 189,A 56.6652,B 1.7184,C -0.0076,E1 1.8105,E2 397.3138} C_DIS
LIN {X 75.1637,Y 110.8686,Z 189,A 55.3267,B 1.7184,C -0.0056,E1 1.8136,E2 398.6438} C_DIS
LIN {X 78.3762,Y 108.6217,Z 189,A 53.7098,B 1.7184,C -0.0029,E1 1.8173,E2 400.2537} C_DIS
LIN {X 81.4086,Y 106.3676,Z 189,A 52.135,B 1.7184,C -0.0002,E1 1.8208,E2 401.8238} C_DIS
LIN {X 84.69,Y 103.774,Z 189,A 50.4436,B 1.7184,C 0.0027,E1 1.8245,E2 403.5038} C_DIS
LIN {X 87.7693,Y 101.1837,Z 189,A 48.7866,B 1.7184,C 0.0057,E1 1.828,E2 405.1535} C_DIS
LIN {X 90.8859,Y 98.3935,Z 189,A 47.1224,B 1.7184,C 0.0086,E1 1.8314,E2 406.8033} C_DIS
LIN {X 93.857,Y 95.563,Z 189,A 45.7049,B 1.7184,C 0.0102,E1 1.8342,E2 408.1815} C_DIS
LIN {X 95.8767,Y 93.5372,Z 189,A 44.3141,B 1.7184,C 0.0138,E1 1.837,E2 409.5921} C_DIS
LIN {X 98.6965,Y 90.5563,Z 189,A 42.6836,B 1.7184,C 0.0168,E1 1.84,E2 411.2082} C_DIS
LIN {X 101.4246,Y 87.4899,Z 189,A 41.0248,B 1.7184,C 0.0201,E1 1.8431,E2 412.8559} C_DIS
LIN {X 104.0576,Y 84.3418,Z 189,A 39.3684,B 1.7183,C 0.0235,E1 1.846,E2 414.501} C_DIS
LIN {X 106.5995,Y 81.1054,Z 189,A 37.6753,B 1.7183,C 0.0271,E1 1.8489,E2 416.1865} C_DIS
LIN {X 109.0846,Y 77.7305,Z 189,A 35.9807,B 1.7182,C 0.0308,E1 1.8516,E2 417.8699} C_DIS
LIN {X 111.3789,Y 74.4055,Z 189,A 34.3777,B 1.7182,C 0.0341,E1 1.8541,E2 419.4585} C_DIS
LIN {X 113.9349,Y 70.4302,Z 189,A 32.5814,B 1.718,C 0.0376,E1 1.8568,E2 421.2286} C_DIS
LIN {X 116.099,Y 66.8025,Z 189,A 30.9107,B 1.718,C 0.0412,E1 1.8591,E2 422.8837} C_DIS
LIN {X 117.7773,Y 63.7973,Z 189,A 29.4125,B 1.7179,C 0.0451,E1 1.8611,E2 424.3854} C_DIS
LIN {X 119.6413,Y 60.2262,Z 189,A 27.9554,B 1.7178,C 0.0478,E1 1.863,E2 425.8112} C_DIS
LIN {X 121.4063,Y 56.5823,Z 189,A 26.3168,B 1.7177,C 0.0516,E1 1.8649,E2 427.4391} C_DIS
LIN {X 123.1108,Y 52.7713,Z 189,A 24.6653,B 1.7176,C 0.0554,E1 1.8668,E2 429.0751} C_DIS
LIN {X 124.6964,Y 48.9068,Z 189,A 23.0378,B 1.7174,C 0.0591,E1 1.8684,E2 430.6841} C_DIS
LIN {X 126.0063,Y 45.4239,Z 189,A 21.5127,B 1.7174,C 0.0629,E1 1.8699,E2 432.2017} C_DIS
LIN {X 127.4141,Y 41.3148,Z 189,A 19.8361,B 1.7172,C 0.0666,E1 1.8714,E2 433.8572} C_DIS
LIN {X 128.5348,Y 37.6793,Z 189,A 18.2729,B 1.717,C 0.0706,E1 1.8726,E2 435.4133} C_DIS
LIN {X 129.5213,Y 34.1368,Z 189,A 16.8767,B 1.7169,C 0.0737,E1 1.8736,E2 436.7887} C_DIS
LIN {X 130.3195,Y 30.9513,Z 189,A 15.5782,B 1.7167,C 0.0769,E1 1.8745,E2 438.0749} C_DIS
LIN {X 131.0396,Y 27.7466,Z 189,A 14.28,B 1.7166,C 0.08,E1 1.8753,E2 439.3607} C_DIS
LIN {X 131.6842,Y 24.5086,Z 189,A 12.9776,B 1.7164,C 0.0832,E1 1.8759,E2 440.6503} C_DIS
LIN {X 132.1857,Y 21.6356,Z 189,A 11.7812,B 1.7163,C 0.0863,E1 1.8765,E2 441.8411} C_DIS
LIN {X 132.7267,Y 18.0278,Z 189,A 10.2663,B 1.7161,C 0.0903,E1 1.8771,E2 443.3512} C_DIS
LIN {X 133.2279,Y 13.8411,Z 189,A 8.7181,B 1.7159,C 0.0936,E1 1.8776,E2 444.8689} C_DIS
LIN {X 133.5277,Y 10.5764,Z 189,A 7.4128,B 1.7157,C 0.0969,E1 1.8779,E2 446.1631} C_DIS
LIN {X 133.738,Y 7.4645,Z 189,A 6.2055,B 1.7156,C 0.0997,E1 1.8781,E2 447.3554} C_DIS
LIN {X 133.8794,Y 4.1901,Z 189,A 4.8367,B 1.7153,C 0.1034,E1 1.8782,E2 448.7208} C_DIS
LIN {X 133.9452,Y 0.4417,Z 189,A 3.3131,B 1.7151,C 0.1074,E1 1.8782,E2 450.2355} C_DIS
LIN {X 133.909,Y -3.1266,Z 189,A 1.9344,B 1.7149,C 0.1106,E1 1.8782,E2 451.5967} C_DIS
LIN {X 133.7372,Y -7.4799,Z 189,A 0.2912,B 1.7146,C 0.1144,E1 1.878,E2 453.2136} C_DIS
LIN {X 133.5264,Y -10.5915,Z 189,A -0.978,B 1.7144,C 0.1176,E1 1.8777,E2 454.4754} C_DIS
LIN {X 133.2232,Y -13.8843,Z 189,A -2.3138,B 1.7142,C 0.1211,E1 1.8774,E2 455.8022} C_DIS
LIN {X 132.8222,Y -17.2993,Z 189,A -3.6317,B 1.714,C 0.1241,E1 1.8769,E2 457.1019} C_DIS
LIN {X 132.3584,Y -20.5487,Z 189,A -4.9272,B 1.7137,C 0.1273,E1 1.8764,E2 458.3846} C_DIS
LIN {X 131.8151,Y -23.7861,Z 189,A -6.2241,B 1.7135,C 0.1304,E1 1.8758,E2 459.6689} C_DIS
LIN {X 131.1929,Y -27.0091,Z 189,A -7.5221,B 1.7133,C 0.1336,E1 1.8751,E2 460.9544} C_DIS
LIN {X 130.492,Y -30.2152,Z 189,A -8.8225,B 1.713,C 0.1367,E1 1.8743,E2 462.2428} C_DIS
LIN {X 129.7084,Y -33.4201,Z 189,A -10.128,B 1.7128,C 0.1398,E1 1.8734,E2 463.5358} C_DIS
LIN {X 128.8787,Y -36.4883,Z 189,A -11.3991,B 1.7125,C 0.1429,E1 1.8725,E2 464.7966} C_DIS
LIN {X 127.9024,Y -39.7777,Z 189,A -12.748,B 1.7122,C 0.1461,E1 1.8714,E2 466.1314} C_DIS
LIN {X 126.9431,Y -42.7382,Z 189,A -13.9946,B 1.712,C 0.1491,E1 1.8703,E2 467.3682} C_DIS
LIN {X 125.8065,Y -45.9781,Z 189,A -15.3369,B 1.7117,C 0.1522,E1 1.8691,E2 468.6954} C_DIS
LIN {X 124.7015,Y -48.8935,Z 189,A -16.5971,B 1.7114,C 0.1552,E1 1.8678,E2 469.9472} C_DIS
LIN {X 123.1152,Y -52.7609,Z 189,A -18.3813,B 1.711,C 0.1599,E1 1.8659,E2 471.7321} C_DIS
LIN {X 121.4015,Y -56.5927,Z 189,A -19.8974,B 1.7107,C 0.1626,E1 1.8642,E2 473.2137} C_DIS
LIN {X 119.8623,Y -59.7852,Z 189,A -21.3983,B 1.7104,C 0.1664,E1 1.8623,E2 474.7139} C_DIS
LIN {X 118.145,Y -63.1133,Z 189,A -22.8478,B 1.7101,C 0.1695,E1 1.8605,E2 476.1449} C_DIS
LIN {X 116.1403,Y -66.7311,Z 189,A -24.4771,B 1.7097,C 0.173,E1 1.8582,E2 477.7575} C_DIS
LIN {X 114.0333,Y -70.2702,Z 189,A -26.1808,B 1.7093,C 0.1769,E1 1.8558,E2 479.455} C_DIS
LIN {X 111.7851,Y -73.7939,Z 189,A -27.7717,B 1.709,C 0.18,E1 1.8534,E2 481.0218} C_DIS
LIN {X 109.8857,Y -76.5936,Z 189,A -29.2435,B 1.7086,C 0.1836,E1 1.8511,E2 482.4979} C_DIS
LIN {X 107.5688,Y -79.815,Z 189,A -30.7772,B 1.7083,C 0.1865,E1 1.8486,E2 484.0117} C_DIS
LIN {X 105.0852,Y -83.0584,Z 189,A -32.4617,B 1.7079,C 0.1901,E1 1.8457,E2 485.6893} C_DIS
LIN {X 102.215,Y -86.5654,Z 189,A -34.2328,B 1.7075,C 0.1934,E1 1.8426,E2 487.4401} C_DIS
LIN {X 99.4124,Y -89.7702,Z 189,A -35.897,B 1.7072,C 0.1964,E1 1.8395,E2 489.0851} C_DIS
LIN {X 96.6393,Y -92.7489,Z 189,A -37.5588,B 1.7068,C 0.1997,E1 1.8363,E2 490.738} C_DIS
LIN {X 93.8928,Y -95.528,Z 189,A -39.1867,B 1.7064,C 0.2029,E1 1.8331,E2 492.3615} C_DIS
LIN {X 90.8167,Y -98.4571,Z 189,A -40.8737,B 1.7061,C 0.2059,E1 1.8297,E2 494.0329} C_DIS
LIN {X 87.7384,Y -101.2105,Z 189,A -42.542,B 1.7057,C 0.2088,E1 1.8262,E2 495.6895} C_DIS
LIN {X 84.6823,Y -103.7802,Z 189,A -44.1815,B 1.7054,C 0.2117,E1 1.8227,E2 497.3214} C_DIS
LIN {X 81.0864,Y -106.614,Z 189,A -46.0778,B 1.705,C 0.215,E1 1.8185,E2 499.2109} C_DIS
LIN {X 77.718,Y -109.0935,Z 189,A -47.7707,B 1.7046,C 0.2176,E1 1.8147,E2 500.8924} C_DIS
LIN {X 74.4126,Y -111.3741,Z 189,A -49.2676,B 1.7044,C 0.2193,E1 1.8113,E2 502.3615} C_DIS
LIN {X 71.6624,Y -113.1634,Z 189,A -50.602,B 1.7041,C 0.2213,E1 1.8082,E2 503.6878} C_DIS
LIN {X 68.8699,Y -114.8846,Z 189,A -52.0057,B 1.7038,C 0.2236,E1 1.8048,E2 505.0926} C_DIS
LIN {X 65.23,Y -116.9899,Z 189,A -53.6624,B 1.7036,C 0.2256,E1 1.8008,E2 506.7317} C_DIS
LIN {X 61.6861,Y -118.8955,Z 189,A -55.3174,B 1.7033,C 0.2278,E1 1.7968,E2 508.3792} C_DIS
LIN {X 58.7443,Y -120.3757,Z 189,A -56.7017,B 1.703,C 0.2298,E1 1.7933,E2 509.7612} C_DIS
LIN {X 54.9124,Y -122.1703,Z 189,A -58.3955,B 1.7028,C 0.2316,E1 1.789,E2 511.4408} C_DIS
LIN {X 51.2448,Y -123.7539,Z 189,A -60.0467,B 1.7025,C 0.2336,E1 1.7848,E2 513.0856} C_DIS
LIN {X 47.5629,Y -125.2161,Z 189,A -61.6923,B 1.7023,C 0.2354,E1 1.7805,E2 514.7258} C_DIS
LIN {X 44.4157,Y -126.3665,Z 189,A -63.244,B 1.7019,C 0.2377,E1 1.7764,E2 516.2942} C_DIS
LIN {X 40.4501,Y -127.6903,Z 189,A -64.7961,B 1.7019,C 0.2384,E1 1.7723,E2 517.816} C_DIS
LIN {X 37.3065,Y -128.644,Z 189,A -66.1588,B 1.7017,C 0.2397,E1 1.7686,E2 519.1739} C_DIS
LIN {X 34.1234,Y -129.5249,Z 189,A -67.5303,B 1.7015,C 0.2408,E1 1.765,E2 520.5408} C_DIS
LIN {X 30.938,Y -130.3227,Z 189,A -68.8964,B 1.7013,C 0.2419,E1 1.7612,E2 521.9026} C_DIS
LIN {X 27.7348,Y -131.0421,Z 189,A -70.2644,B 1.7012,C 0.243,E1 1.7575,E2 523.2666} C_DIS
LIN {X 24.515,Y -131.683,Z 189,A -71.6336,B 1.7011,C 0.2439,E1 1.7537,E2 524.632} C_DIS
LIN {X 21.2234,Y -132.2539,Z 189,A -73.0499,B 1.7009,C 0.2449,E1 1.7498,E2 526.0475} C_DIS
LIN {X 17.9941,Y -132.7312,Z 189,A -74.421,B 1.7009,C 0.2456,E1 1.746,E2 527.416} C_DIS
LIN {X 14.7472,Y -133.1304,Z 189,A -75.7948,B 1.7007,C 0.2464,E1 1.7422,E2 528.7871} C_DIS
LIN {X 11.1956,Y -133.4754,Z 189,A -77.3601,B 1.7006,C 0.2473,E1 1.7378,E2 530.3585} C_DIS
LIN {X 7.4796,Y -133.7372,Z 189,A -78.9366,B 1.7005,C 0.248,E1 1.7334,E2 531.9336} C_DIS
LIN {X 4.1759,Y -133.8798,Z 189,A -80.3814,B 1.7004,C 0.2486,E1 1.7294,E2 533.3831} C_DIS
LIN {X 0.9696,Y -133.9381,Z 189,A -81.273,B 1.7006,C 0.247,E1 1.727,E2 534.2109} C_DIS
Enddeposition()
LIN {X 0.9696,Y -133.9381,Z 189,A -81.2731,B 1.7006,C 0.247,E1 1.727,E2 534.211} C_DIS
Startdeposition()
$VEL.CP = VEL_PRINT
LIN {X 1.7185,Y -134.8334,Z 189,A -80.6184,B 1.7009,C 0.2463,E1 1.7291,E2 533.5386} C_DIS
LIN {X 8.6039,Y -134.5688,Z 189,A -77.7142,B 1.701,C 0.2452,E1 1.7372,E2 530.6362} C_DIS
LIN {X 12.7324,Y -134.2408,Z 189,A -76.005,B 1.7011,C 0.2445,E1 1.742,E2 528.933} C_DIS
LIN {X 15.6816,Y -133.9285,Z 189,A -74.278,B 1.7015,C 0.2416,E1 1.747,E2 527.1415} C_DIS
LIN {X 20.1814,Y -133.325,Z 189,A -72.6989,B 1.7015,C 0.242,E1 1.7512,E2 525.6092} C_DIS
LIN {X 24.9941,Y -132.5068,Z 189,A -70.8401,B 1.7015,C 0.2415,E1 1.7563,E2 523.7785} C_DIS
LIN {X 28.6524,Y -131.7639,Z 189,A -69.3024,B 1.7017,C 0.2404,E1 1.7605,E2 522.2464} C_DIS
LIN {X 32.0829,Y -130.9716,Z 189,A -67.7526,B 1.7019,C 0.2388,E1 1.7647,E2 520.6884} C_DIS
LIN {X 36.009,Y -129.9464,Z 189,A -66.1889,B 1.7021,C 0.2379,E1 1.7689,E2 519.1454} C_DIS
LIN {X 39.2991,Y -128.9892,Z 189,A -64.778,B 1.7022,C 0.2366,E1 1.7727,E2 517.7396} C_DIS
LIN {X 42.6528,Y -127.9193,Z 189,A -63.4892,B 1.7023,C 0.2361,E1 1.776,E2 516.478} C_DIS
LIN {X 47.0889,Y -126.3538,Z 189,A -61.4293,B 1.7027,C 0.2334,E1 1.7815,E2 514.4085} C_DIS
LIN {X 50.1436,Y -125.173,Z 189,A -59.1308,B 1.7036,C 0.2267,E1 1.7878,E2 511.9853} C_DIS
LIN {X 56.436,Y -122.4646,Z 189,A -57.2317,B 1.7034,C 0.2284,E1 1.7923,E2 510.2223} C_DIS
LIN {X 59.9989,Y -120.7594,Z 189,A -55.5957,B 1.7037,C 0.2262,E1 1.7964,E2 508.5909} C_DIS
LIN {X 63.7979,Y -118.7979,Z 189,A -53.8296,B 1.704,C 0.2237,E1 1.8008,E2 506.8303} C_DIS
LIN {X 66.4602,Y -117.3299,Z 189,A -52.3852,B 1.7044,C 0.2208,E1 1.8043,E2 505.3644} C_DIS
LIN {X 69.2949,Y -115.678,Z 189,A -51.2926,B 1.7044,C 0.2203,E1 1.8069,E2 504.3116} C_DIS
LIN {X 72.9419,Y -113.4137,Z 189,A -49.6002,B 1.7047,C 0.218,E1 1.8108,E2 502.6356} C_DIS
LIN {X 75.8416,Y -111.4955,Z 189,A -48.0953,B 1.7051,C 0.2153,E1 1.8143,E2 501.1258} C_DIS
LIN {X 79.4349,Y -108.9649,Z 189,A -46.3569,B 1.7054,C 0.2127,E1 1.8183,E2 499.4034} C_DIS
LIN {X 84.6304,Y -104.98,Z 189,A -42.8881,B 1.7066,C 0.2032,E1 1.8261,E2 495.8397} C_DIS
LIN {X 89.8197,Y -100.5762,Z 189,A -41.1695,B 1.7064,C 0.2048,E1 1.8294,E2 494.2771} C_DIS
LIN {X 94.2905,Y -96.3973,Z 189,A -38.5101,B 1.707,C 0.1991,E1 1.8348,E2 491.6079} C_DIS
LIN {X 100.2404,Y -90.1946,Z 189,A -35.352,B 1.7076,C 0.1944,E1 1.8408,E2 488.5131} C_DIS
LIN {X 103.8248,Y -86.0437,Z 189,A -32.8953,B 1.7083,C 0.1884,E1 1.8452,E2 486.0379} C_DIS
LIN {X 106.2558,Y -83.0237,Z 189,A -30.4801,B 1.7092,C 0.1796,E1 1.8496,E2 483.5187} C_DIS
LIN {X 110.517,Y -77.2604,Z 189,A -28.3832,B 1.7093,C 0.1786,E1 1.8528,E2 481.5464} C_DIS
LIN {X 113.1596,Y -73.335,Z 189,A -26.6929,B 1.7096,C 0.1759,E1 1.8553,E2 479.8969} C_DIS
LIN {X 115.1202,Y -70.218,Z 189,A -25.2408,B 1.7099,C 0.1728,E1 1.8574,E2 478.4585} C_DIS
LIN {X 117.2561,Y -66.5897,Z 189,A -23.5372,B 1.7103,C 0.1689,E1 1.8598,E2 476.7647} C_DIS
LIN {X 119.837,Y -61.8239,Z 189,A -21.3292,B 1.7108,C 0.1638,E1 1.8627,E2 474.5675} C_DIS
LIN {X 121.5193,Y -58.4444,Z 189,A -19.8837,B 1.7111,C 0.1607,E1 1.8644,E2 473.1415} C_DIS
LIN {X 123.0324,Y -55.1871,Z 189,A -18.5125,B 1.7114,C 0.1578,E1 1.866,E2 471.7895} C_DIS
LIN {X 124.8961,Y -50.8306,Z 189,A -16.6244,B 1.7118,C 0.1534,E1 1.868,E2 469.9163} C_DIS
LIN {X 126.2473,Y -47.3731,Z 189,A -15.2704,B 1.712,C 0.1507,E1 1.8693,E2 468.5902} C_DIS
LIN {X 127.3158,Y -44.4223,Z 189,A -13.9008,B 1.7123,C 0.1469,E1 1.8706,E2 467.215} C_DIS
LIN {X 129.6092,Y -37.2098,Z 189,A -10.9374,B 1.7129,C 0.14,E1 1.873,E2 464.2822} C_DIS
LIN {X 130.5537,Y -33.7445,Z 189,A -9.4718,B 1.7132,C 0.1362,E1 1.8741,E2 462.8234} C_DIS
LIN {X 131.4405,Y -30.1004,Z 189,A -8.0798,B 1.7134,C 0.1333,E1 1.8749,E2 461.4563} C_DIS
LIN {X 132.2124,Y -26.5078,Z 189,A -6.6118,B 1.7137,C 0.1296,E1 1.8758,E2 459.9993} C_DIS
LIN {X 132.9433,Y -22.558,Z 189,A -5.1579,B 1.7139,C 0.1266,E1 1.8765,E2 458.5768} C_DIS
LIN {X 133.4695,Y -19.1986,Z 189,A -3.6734,B 1.7142,C 0.1224,E1 1.8771,E2 457.0861} C_DIS
LIN {X 133.9813,Y -15.2396,Z 189,A -1.8916,B 1.7146,C 0.117,E1 1.8777,E2 455.2924} C_DIS
LIN {X 134.308,Y -12.0211,Z 189,A -0.7784,B 1.7148,C 0.115,E1 1.878,E2 454.2118} C_DIS
LIN {X 134.589,Y -8.2767,Z 189,A 0.6311,B 1.715,C 0.1118,E1 1.8782,E2 452.825} C_DIS
LIN {X 134.8138,Y -2.8961,Z 189,A 2.8154,B 1.7153,C 0.1061,E1 1.8784,E2 450.6526} C_DIS
LIN {X 134.8455,Y 0.2376,Z 189,A 4.1724,B 1.7156,C 0.1022,E1 1.8784,E2 449.2917} C_DIS
LIN {X 134.7518,Y 4.9754,Z 189,A 5.8077,B 1.7157,C 0.0992,E1 1.8783,E2 447.7031} C_DIS
LIN {X 134.5539,Y 8.8472,Z 189,A 7.3989,B 1.716,C 0.095,E1 1.878,E2 446.1181} C_DIS
LIN {X 134.3057,Y 12.0482,Z 189,A 8.7677,B 1.7162,C 0.0911,E1 1.8777,E2 444.748} C_DIS
LIN {X 133.7553,Y 17.0988,Z 189,A 10.6293,B 1.7164,C 0.0872,E1 1.8771,E2 442.9227} C_DIS
LIN {X 133.1771,Y 21.1374,Z 189,A 12.2682,B 1.7166,C 0.083,E1 1.8764,E2 441.2948} C_DIS
LIN {X 132.3793,Y 25.6613,Z 189,A 14.0551,B 1.7168,C 0.0787,E1 1.8755,E2 439.5275} C_DIS
LIN {X 131.511,Y 29.7916,Z 189,A 15.6311,B 1.717,C 0.0753,E1 1.8746,E2 437.9778} C_DIS
LIN {X 130.7489,Y 32.9756,Z 189,A 16.7996,B 1.717,C 0.073,E1 1.8738,E2 436.8362} C_DIS
LIN {X 129.9534,Y 35.9842,Z 189,A 18.1718,B 1.7172,C 0.069,E1 1.8728,E2 435.4573} C_DIS
LIN {X 128.9559,Y 39.4079,Z 189,A 19.5151,B 1.7173,C 0.0661,E1 1.8718,E2 434.1346} C_DIS
LIN {X 128.1024,Y 42.1027,Z 189,A 20.7376,B 1.7175,C 0.0627,E1 1.8707,E2 432.909} C_DIS
LIN {X 126.9553,Y 45.4428,Z 189,A 22.2566,B 1.7176,C 0.0586,E1 1.8693,E2 431.3871} C_DIS
LIN {X 125.2678,Y 49.9085,Z 189,A 24.0244,B 1.7177,C 0.055,E1 1.8675,E2 429.6508} C_DIS
LIN {X 123.8956,Y 53.2218,Z 189,A 25.3263,B 1.7178,C 0.0524,E1 1.8661,E2 428.3755} C_DIS
LIN {X 122.4471,Y 56.4738,Z 189,A 26.9496,B 1.7179,C 0.0478,E1 1.8642,E2 426.7382} C_DIS
LIN {X 120.3088,Y 60.8969,Z 189,A 28.6615,B 1.718,C 0.0449,E1 1.8622,E2 425.0715} C_DIS
LIN {X 118.5718,Y 64.2184,Z 189,A 30.2914,B 1.7181,C 0.0406,E1 1.86,E2 423.4367} C_DIS
LIN {X 116.6768,Y 67.5991,Z 189,A 31.875,B 1.7182,C 0.037,E1 1.8578,E2 421.8604} C_DIS
LIN {X 114.1578,Y 71.7716,Z 189,A 33.7459,B 1.7182,C 0.0332,E1 1.8551,E2 420.0132} C_DIS
LIN {X 112.0583,Y 75.0072,Z 189,A 35.4579,B 1.7184,C 0.0288,E1 1.8525,E2 418.2919} C_DIS
LIN {X 110.1905,Y 77.7249,Z 189,A 36.5659,B 1.7184,C 0.0273,E1 1.8507,E2 417.2192} C_DIS
LIN {X 107.4875,Y 81.4225,Z 189,A 38.3935,B 1.7184,C 0.0235,E1 1.8477,E2 415.4055} C_DIS
LIN {X 104.6901,Y 84.9898,Z 189,A 40.2306,B 1.7184,C 0.0196,E1 1.8445,E2 413.5789} C_DIS
LIN {X 101.8075,Y 88.4219,Z 189,A 42.0072,B 1.7185,C 0.0162,E1 1.8413,E2 411.8172} C_DIS
LIN {X 98.9155,Y 91.6458,Z 189,A 43.7466,B 1.7185,C 0.0128,E1 1.8381,E2 410.0897} C_DIS
LIN {X 95.7866,Y 94.9109,Z 189,A 45.532,B 1.7185,C 0.0095,E1 1.8346,E2 408.3204} C_DIS
LIN {X 93.2113,Y 97.4411,Z 189,A 46.9609,B 1.7185,C 0.0069,E1 1.8318,E2 406.9038} C_DIS
LIN {X 89.8203,Y 100.5757,Z 189,A 48.8213,B 1.7186,C 0.0036,E1 1.8279,E2 405.0554} C_DIS
LIN {X 86.4385,Y 103.4968,Z 189,A 50.5854,B 1.7186,C 0.0007,E1 1.8242,E2 403.3073} C_DIS
LIN {X 83.0201,Y 106.2586,Z 189,A 52.3933,B 1.7186,C -0.0025,E1 1.8203,E2 401.5063} C_DIS
LIN {X 79.5326,Y 108.8936,Z 189,A 54.1708,B 1.7186,C -0.0055,E1 1.8163,E2 399.7382} C_DIS
LIN {X 76.0405,Y 111.36,Z 189,A 55.8083,B 1.7186,C -0.0077,E1 1.8126,E2 398.1219} C_DIS
LIN {X 73.7895,Y 112.8646,Z 189,A 57.0275,B 1.7186,C -0.01,E1 1.8097,E2 396.8946} C_DIS
LIN {X 69.8314,Y 115.3546,Z 189,A 58.8385,B 1.7186,C -0.0123,E1 1.8054,E2 395.1044} C_DIS
LIN {X 66.2458,Y 117.4506,Z 189,A 60.5111,B 1.7186,C -0.0146,E1 1.8014,E2 393.4427} C_DIS
LIN {X 61.7051,Y 119.8974,Z 189,A 62.6113,B 1.7186,C -0.0174,E1 1.7962,E2 391.3535} C_DIS
LIN {X 58.4444,Y 121.5193,Z 189,A 64.007,B 1.7186,C -0.0189,E1 1.7927,E2 389.9756} C_DIS
LIN {X 55.501,Y 122.892,Z 189,A 65.2608,B 1.7185,C -0.0201,E1 1.7896,E2 388.7367} C_DIS
LIN {X 52.2744,Y 124.2984,Z 189,A 66.7274,B 1.7185,C -0.0219,E1 1.7858,E2 387.2738} C_DIS
LIN {X 49.0552,Y 125.6034,Z 189,A 68.2467,B 1.7185,C -0.024,E1 1.7819,E2 385.7496} C_DIS
LIN {X 46.1586,Y 126.6972,Z 189,A 69.4333,B 1.7185,C -0.0249,E1 1.7788,E2 384.5783} C_DIS
LIN {X 40.8678,Y 128.5008,Z 189,A 71.8331,B 1.7184,C -0.0277,E1 1.7724,E2 382.1761} C_DIS
LIN {X 36.7711,Y 129.7333,Z 189,A 73.5548,B 1.7184,C -0.0291,E1 1.7678,E2 380.4661} C_DIS
LIN {X 33.3835,Y 130.6454,Z 189,A 75.0736,B 1.7184,C -0.0306,E1 1.7637,E2 378.9443} C_DIS
LIN {X 29.2301,Y 131.6392,Z 189,A 76.9257,B 1.7184,C -0.0323,E1 1.7586,E2 377.0885} C_DIS
LIN {X 25.5192,Y 132.4064,Z 189,A 78.3138,B 1.7183,C -0.0326,E1 1.7549,E2 375.7264} C_DIS
LIN {X 22.1849,Y 133.0056,Z 189,A 79.5373,B 1.7183,C -0.0327,E1 1.7516,E2 374.5282} C_DIS
LIN {X 19.3775,Y 133.4439,Z 189,A 81.0161,B 1.7183,C -0.0346,E1 1.7474,E2 373.0186} C_DIS
LIN {X 15.4581,Y 133.9552,Z 189,A 82.6277,B 1.7183,C -0.0353,E1 1.7429,E2 371.4153} C_DIS
LIN {X 11.7727,Y 134.329,Z 189,A 84.1704,B 1.7183,C -0.036,E1 1.7386,E2 369.8769} C_DIS
LIN {X 8.2934,Y 134.588,Z 189,A 85.6276,B 1.7183,C -0.0366,E1 1.7345,E2 368.4231} C_DIS
LIN {X 3.9676,Y 134.7851,Z 189,A 87.5367,B 1.7183,C -0.0375,E1 1.7292,E2 366.5067} C_DIS
LIN {X -0.6877,Y 134.8416,Z 189,A 89.3978,B 1.7182,C -0.0375,E1 1.724,E2 364.6598} C_DIS
LIN {X -5.0019,Y 134.7507,Z 189,A 91.1913,B 1.7182,C -0.0377,E1 1.719,E2 362.8717} C_DIS
LIN {X -8.1133,Y 134.5991,Z 189,A 92.6429,B 1.7182,C -0.0383,E1 1.7149,E2 361.406} C_DIS
LIN {X -12.7418,Y 134.2399,Z 189,A 94.5529,B 1.7182,C -0.0381,E1 1.7096,E2 359.5041} C_DIS
LIN {X -16.857,Y 133.787,Z 189,A 96.4031,B 1.7182,C -0.0383,E1 1.7044,E2 357.6443} C_DIS
LIN {X -20.3887,Y 133.293,Z 189,A 98.2459,B 1.7182,C -0.0391,E1 1.6992,E2 355.7644} C_DIS
LIN {X -24.4425,Y 132.6111,Z 189,A 99.5846,B 1.7182,C -0.0373,E1 1.6956,E2 354.4737} C_DIS
LIN {X -28.2904,Y 131.842,Z 189,A 101.2994,B 1.7182,C -0.0369,E1 1.6909,E2 352.7542} C_DIS
LIN {X -32.3842,Y 130.8989,Z 189,A 103.0956,B 1.7182,C -0.0362,E1 1.686,E2 350.9577} C_DIS
LIN {X -36.1291,Y 129.9128,Z 189,A 104.7181,B 1.7182,C -0.0353,E1 1.6816,E2 349.3386} C_DIS
LIN {X -39.096,Y 129.0514,Z 189,A 105.9977,B 1.7182,C -0.0345,E1 1.6782,E2 348.0636} C_DIS
LIN {X -41.9889,Y 128.1404,Z 189,A 107.67,B 1.7182,C -0.0347,E1 1.6736,E2 346.3479} C_DIS
LIN {X -45.0665,Y 127.0909,Z 189,A 108.8167,B 1.7182,C -0.0331,E1 1.6706,E2 345.2291} C_DIS
LIN {X -48.3507,Y 125.8773,Z 189,A 110.3844,B 1.7183,C -0.0322,E1 1.6665,E2 343.6529} C_DIS
LIN {X -51.6855,Y 124.5443,Z 189,A 111.6805,B 1.7183,C -0.0304,E1 1.6632,E2 342.3841} C_DIS
LIN {X -54.44,Y 123.3666,Z 189,A 113.1573,B 1.7183,C -0.0297,E1 1.6593,E2 340.8847} C_DIS
LIN {X -57.4398,Y 121.9992,Z 189,A 114.7884,B 1.7183,C -0.0289,E1 1.6551,E2 339.2279} C_DIS
LIN {X -60.7031,Y 120.4075,Z 189,A 116.2121,B 1.7183,C -0.027,E1 1.6516,E2 337.8188} C_DIS
LIN {X -64.1174,Y 118.6263,Z 189,A 118.1769,B 1.7184,C -0.0259,E1 1.6467,E2 335.8171} C_DIS
LIN {X -68.6248,Y 116.0771,Z 189,A 120.2767,B 1.7184,C -0.023,E1 1.6416,E2 333.7303} C_DIS
LIN {X -71.0787,Y 114.5905,Z 189,A 121.7412,B 1.7184,C -0.022,E1 1.638,E2 332.2381} C_DIS
LIN {X -75.4947,Y 111.7304,Z 189,A 123.872,B 1.7185,C -0.0187,E1 1.6331,E2 330.1208} C_DIS
LIN {X -79.0088,Y 109.2737,Z 189,A 125.5937,B 1.7185,C -0.0159,E1 1.6292,E2 328.4121} C_DIS
LIN {X -82.6321,Y 106.5601,Z 189,A 127.7649,B 1.7185,C -0.0134,E1 1.6243,E2 326.2133} C_DIS
LIN {X -85.9032,Y 103.9411,Z 189,A 129.6608,B 1.7185,C -0.0107,E1 1.6201,E2 324.3052} C_DIS
LIN {X -89.0984,Y 101.2159,Z 189,A 131.5969,B 1.7185,C -0.0079,E1 1.616,E2 322.3525} C_DIS
LIN {X -92.7245,Y 97.9048,Z 189,A 133.8679,B 1.7186,C -0.0045,E1 1.6113,E2 320.0612} C_DIS
LIN {X -96.279,Y 94.4111,Z 189,A 135.968,B 1.7186,C -0.0006,E1 1.6072,E2 317.9646} C_DIS
LIN {X -99.2564,Y 91.2758,Z 189,A 137.9366,B 1.7186,C 0.0028,E1 1.6034,E2 315.9818} C_DIS
LIN {X -102.2935,Y 87.8589,Z 189,A 140.0573,B 1.7186,C 0.0064,E1 1.5994,E2 313.8415} C_DIS
LIN {X -105.2381,Y 84.3104,Z 189,A 142.1332,B 1.7186,C 0.0104,E1 1.5957,E2 311.7532} C_DIS
LIN {X -107.7678,Y 81.051,Z 189,A 143.9228,B 1.7186,C 0.0141,E1 1.5927,E2 309.9605} C_DIS
LIN {X -110.2879,Y 77.5868,Z 189,A 145.8415,B 1.7186,C 0.0179,E1 1.5896,E2 308.0313} C_DIS
LIN {X -112.382,Y 74.5222,Z 189,A 147.653,B 1.7185,C 0.0212,E1 1.5867,E2 306.193} C_DIS
LIN {X -114.7684,Y 70.7916,Z 189,A 149.6036,B 1.7185,C 0.0255,E1 1.5838,E2 304.2355} C_DIS
LIN {X -116.814,Y 67.3622,Z 189,A 151.3896,B 1.7184,C 0.0294,E1 1.5812,E2 302.44} C_DIS
LIN {X -118.7828,Y 63.8259,Z 189,A 153.385,B 1.7183,C 0.0333,E1 1.5785,E2 300.4127} C_DIS
LIN {X -120.7942,Y 59.9284,Z 189,A 155.2147,B 1.7182,C 0.0379,E1 1.5762,E2 298.5883} C_DIS
LIN {X -122.0458,Y 57.3417,Z 189,A 156.545,B 1.7182,C 0.0408,E1 1.5746,E2 297.2458} C_DIS
LIN {X -123.816,Y 53.4058,Z 189,A 158.4596,B 1.718,C 0.0454,E1 1.5724,E2 295.3226} C_DIS
LIN {X -125.0231,Y 50.5156,Z 189,A 159.9732,B 1.718,C 0.0486,E1 1.5708,E2 293.7878} C_DIS
LIN {X -126.1252,Y 47.699,Z 189,A 161.3982,B 1.7178,C 0.0519,E1 1.5694,E2 292.3468} C_DIS
LIN {X -127.2661,Y 44.5659,Z 189,A 162.9822,B 1.7178,C 0.0554,E1 1.5679,E2 290.7434} C_DIS
LIN {X -128.5281,Y 40.7823,Z 189,A 164.7862,B 1.7176,C 0.0598,E1 1.5663,E2 288.9272} C_DIS
LIN {X -129.7285,Y 36.7883,Z 189,A 166.7469,B 1.7174,C 0.0645,E1 1.5647,E2 286.9447} C_DIS
LIN {X -130.7265,Y 33.0637,Z 189,A 169.2034,B 1.7172,C 0.0683,E1 1.563,E2 284.3884} C_DIS
LIN {X -131.9317,Y 27.8749,Z 189,A 171.081,B 1.717,C 0.0748,E1 1.5619,E2 282.5601} C_DIS
LIN {X -132.6984,Y 23.955,Z 189,A 172.783,B 1.7168,C 0.0794,E1 1.561,E2 280.8586} C_DIS
LIN {X -133.2194,Y 20.864,Z 189,A 174.2502,B 1.7166,C 0.083,E1 1.5604,E2 279.3755} C_DIS
LIN {X -133.7407,Y 17.2103,Z 189,A 176.0518,B 1.7164,C 0.0872,E1 1.5597,E2 277.5459} C_DIS
LIN {X -134.2173,Y 12.9778,Z 189,A 177.8892,B 1.7161,C 0.0923,E1 1.5591,E2 275.7062} C_DIS
LIN {X -134.5095,Y 9.4876,Z 189,A 179.6454,B 1.7159,C 0.0963,E1 1.5588,E2 273.9175} C_DIS
LIN {X -134.7395,Y 5.2898,Z 189,A -178.4516,B 1.7156,C 0.1012,E1 1.5585,E2 272.001} C_DIS
LIN {X -134.8422,Y 0.7527,Z 189,A -176.4119,B 1.7153,C 0.1065,E1 1.5585,E2 269.9485} C_DIS
LIN {X -134.8069,Y -3.1838,Z 189,A -174.4715,B 1.715,C 0.111,E1 1.5585,E2 267.9754} C_DIS
LIN {X -134.6643,Y -6.948,Z 189,A -172.8094,B 1.7147,C 0.1155,E1 1.5587,E2 266.3065} C_DIS
LIN {X -134.3861,Y -11.0965,Z 189,A -170.87,B 1.7144,C 0.1203,E1 1.5591,E2 264.3462} C_DIS
LIN {X -134.0376,Y -14.7201,Z 189,A -169.1301,B 1.7141,C 0.1245,E1 1.5596,E2 262.5826} C_DIS
LIN {X -133.4922,Y -19.0392,Z 189,A -167.1686,B 1.7137,C 0.1295,E1 1.5604,E2 260.6079} C_DIS
LIN {X -132.8528,Y -23.0919,Z 189,A -165.1555,B 1.7134,C 0.1341,E1 1.5613,E2 258.5613} C_DIS
LIN {X -132.1516,Y -26.8067,Z 189,A -163.5966,B 1.713,C 0.1385,E1 1.5621,E2 257.0093} C_DIS
LIN {X -131.4674,Y -29.9828,Z 189,A -162.1088,B 1.7127,C 0.1422,E1 1.563,E2 255.5084} C_DIS
LIN {X -130.8224,Y -32.6861,Z 189,A -160.8504,B 1.7125,C 0.1453,E1 1.5639,E2 254.2407} C_DIS
LIN {X -129.5788,Y -37.3136,Z 189,A -158.634,B 1.712,C 0.1506,E1 1.5656,E2 252.0021} C_DIS
LIN {X -128.7102,Y -40.2103,Z 189,A -156.5401,B 1.7118,C 0.1533,E1 1.5674,E2 249.804} C_DIS
LIN {X -127.2686,Y -44.5586,Z 189,A -154.6111,B 1.7113,C 0.1584,E1 1.5692,E2 247.878} C_DIS
LIN {X -125.938,Y -48.1946,Z 189,A -153.1415,B 1.7109,C 0.1628,E1 1.5706,E2 246.432} C_DIS
LIN {X -124.509,Y -51.7699,Z 189,A -151.489,B 1.7105,C 0.1669,E1 1.5723,E2 244.778} C_DIS
LIN {X -123.1515,Y -54.921,Z 189,A -149.8724,B 1.7101,C 0.1704,E1 1.5742,E2 243.1412} C_DIS
LIN {X -121.6172,Y -58.2394,Z 189,A -148.3247,B 1.7098,C 0.1743,E1 1.576,E2 241.5949} C_DIS
LIN {X -120.2826,Y -60.9484,Z 189,A -146.9547,B 1.7094,C 0.1773,E1 1.5777,E2 240.2139} C_DIS
LIN {X -118.4642,Y -64.4157,Z 189,A -145.0312,B 1.7091,C 0.181,E1 1.5803,E2 238.257} C_DIS
LIN {X -116.6114,Y -67.712,Z 189,A -143.3044,B 1.7087,C 0.1846,E1 1.5827,E2 236.515} C_DIS
LIN {X -114.6373,Y -71.0035,Z 189,A -141.5421,B 1.7083,C 0.1882,E1 1.5853,E2 234.7358} C_DIS
LIN {X -112.6047,Y -74.1842,Z 189,A -139.7809,B 1.7079,C 0.1916,E1 1.588,E2 232.9543} C_DIS
LIN {X -110.117,Y -77.8291,Z 189,A -137.8051,B 1.7075,C 0.1955,E1 1.5912,E2 230.9656} C_DIS
LIN {X -107.6351,Y -81.2267,Z 189,A -135.8644,B 1.707,C 0.1991,E1 1.5945,E2 229.005} C_DIS
LIN {X -104.9967,Y -84.6097,Z 189,A -133.9165,B 1.7066,C 0.2027,E1 1.5979,E2 227.0408} C_DIS
LIN {X -102.1715,Y -88.0005,Z 189,A -131.9042,B 1.7062,C 0.2062,E1 1.6016,E2 225.0106} C_DIS
LIN {X -99.0858,Y -91.4614,Z 189,A -129.6483,B 1.7058,C 0.2095,E1 1.6059,E2 222.7169} C_DIS
LIN {X -93.5138,Y -97.1516,Z 189,A -125.6898,B 1.7052,C 0.2145,E1 1.6139,E2 218.6816} C_DIS
LIN {X -89.9269,Y -100.4802,Z 189,A -124.0452,B 1.7046,C 0.219,E1 1.6172,E2 217.0956} C_DIS
LIN {X -86.4734,Y -103.4675,Z 189,A -122.004,B 1.7042,C 0.2219,E1 1.6216,E2 215.0408} C_DIS
LIN {X -82.9433,Y -106.3188,Z 189,A -119.9544,B 1.7039,C 0.2246,E1 1.6261,E2 212.9749} C_DIS
LIN {X -79.4796,Y -108.9325,Z 189,A -118.0319,B 1.7035,C 0.2272,E1 1.6305,E2 211.0419} C_DIS
LIN {X -75.595,Y -111.6624,Z 189,A -115.9714,B 1.7032,C 0.2298,E1 1.6352,E2 208.9754} C_DIS
LIN {X -72.0132,Y -114.0053,Z 189,A -114.0805,B 1.7029,C 0.232,E1 1.6397,E2 207.0746} C_DIS
LIN {X -68.4067,Y -116.2052,Z 189,A -112.3749,B 1.7025,C 0.2345,E1 1.6438,E2 205.3809} C_DIS
LIN {X -64.6536,Y -118.3344,Z 189,A -110.3623,B 1.7023,C 0.2361,E1 1.6488,E2 203.3439} C_DIS
LIN {X -61.4286,Y -120.0382,Z 189,A -108.7708,B 1.7021,C 0.2376,E1 1.6527,E2 201.7465} C_DIS
LIN {X -58.421,Y -121.5305,Z 189,A -107.5232,B 1.7018,C 0.2395,E1 1.6558,E2 200.5228} C_DIS
LIN {X -55.7377,Y -122.7862,Z 189,A -105.9141,B 1.7018,C 0.2397,E1 1.66,E2 198.8662} C_DIS
LIN {X -52.4473,Y -124.2261,Z 189,A -104.3708,B 1.7016,C 0.2409,E1 1.664,E2 197.3201} C_DIS
LIN {X -49.2694,Y -125.5202,Z 189,A -102.9309,B 1.7015,C 0.2421,E1 1.6678,E2 195.8823} C_DIS
LIN {X -44.1283,Y -127.4178,Z 189,A -100.6032,B 1.7012,C 0.2438,E1 1.6739,E2 193.5542} C_DIS
LIN {X -41.1341,Y -128.4157,Z 189,A -99.2463,B 1.7012,C 0.2445,E1 1.6775,E2 192.1947} C_DIS
LIN {X -38.0481,Y -129.3637,Z 189,A -97.8278,B 1.701,C 0.2451,E1 1.6813,E2 190.7696} C_DIS
LIN {X -34.4306,Y -130.3735,Z 189,A -96.1782,B 1.701,C 0.2457,E1 1.6858,E2 189.1122} C_DIS
LIN {X -30.2407,Y -131.4085,Z 189,A -94.3171,B 1.7009,C 0.2463,E1 1.6909,E2 187.2467} C_DIS
LIN {X -26.5403,Y -132.2058,Z 189,A -92.7222,B 1.7009,C 0.2468,E1 1.6953,E2 185.653} C_DIS
LIN {X -21.7662,Y -133.0754,Z 189,A -90.5235,B 1.7009,C 0.2468,E1 1.7014,E2 183.435} C_DIS
LIN {X -17.5967,Y -133.6901,Z 189,A -88.7814,B 1.7008,C 0.2471,E1 1.7062,E2 181.6987} C_DIS
LIN {X -13.1228,Y -134.2033,Z 189,A -86.9922,B 1.7007,C 0.2477,E1 1.7112,E2 179.9257} C_DIS
LIN {X -9.6834,Y -134.4952,Z 189,A -85.1889,B 1.7009,C 0.2462,E1 1.7164,E2 178.0758} C_DIS
LIN {X -6.3886,Y -134.6924,Z 189,A -84.0897,B 1.7007,C 0.2473,E1 1.7193,E2 177.0173} C_DIS
LIN {X -1.8671,Y -134.8309,Z 189,A -81.8289,B 1.701,C 0.2454,E1 1.7258,E2 174.7094} C_DIS
LIN {X -1.8671,Y -134.8309,Z 189,A -81.8289,B 1.701,C 0.2454,E1 1.7258,E2 174.7094} C_DIS
Enddeposition()
LIN {X 0.957,Y -135.7293,Z 189,A -82.297,B 1.6996,C 0.2531,E1 1.7235,E2 175.4318} C_DIS
Startdeposition()
$VEL.CP = VEL_PRINT
LIN {X -5.0519,Y -135.6486,Z 189,A -83.8903,B 1.7001,C 0.2496,E1 1.7194,E2 176.8987} C_DIS
LIN {X -11.8006,Y -135.229,Z 189,A -87.0051,B 1.6999,C 0.251,E1 1.7106,E2 180.0505} C_DIS
LIN {X -15.821,Y -134.8174,Z 189,A -88.7038,B 1.6999,C 0.2509,E1 1.7058,E2 181.749} C_DIS
LIN {X -19.3912,Y -134.3502,Z 189,A -90.2117,B 1.6999,C 0.2507,E1 1.7016,E2 183.2559} C_DIS
LIN {X -24.9735,Y -133.4262,Z 189,A -92.6718,B 1.6999,C 0.2504,E1 1.6948,E2 185.7266} C_DIS
LIN {X -28.6545,Y -132.6833,Z 189,A -94.2083,B 1.7001,C 0.2498,E1 1.6906,E2 187.2571} C_DIS
LIN {X -32.16,Y -131.8779,Z 189,A -95.7416,B 1.7001,C 0.2493,E1 1.6864,E2 188.7929} C_DIS
LIN {X -36.2264,Y -130.8193,Z 189,A -97.5736,B 1.7003,C 0.2487,E1 1.6814,E2 190.6334} C_DIS
LIN {X -39.7279,Y -129.7983,Z 189,A -99.1035,B 1.7003,C 0.2478,E1 1.6773,E2 192.1625} C_DIS
LIN {X -42.8361,Y -128.8059,Z 189,A -100.4655,B 1.7005,C 0.2469,E1 1.6737,E2 193.5228} C_DIS
LIN {X -46.172,Y -127.6482,Z 189,A -102.0154,B 1.7006,C 0.2461,E1 1.6696,E2 195.0812} C_DIS
LIN {X -51.5548,Y -125.5733,Z 189,A -104.4909,B 1.7009,C 0.2443,E1 1.6631,E2 197.5628} C_DIS
LIN {X -54.6524,Y -124.2563,Z 189,A -106.3966,B 1.7009,C 0.2446,E1 1.658,E2 199.5343} C_DIS
LIN {X -58.1478,Y -122.6575,Z 189,A -107.4593,B 1.7013,C 0.2414,E1 1.6555,E2 200.5217} C_DIS
LIN {X -62.0505,Y -120.7306,Z 189,A -109.6034,B 1.7014,C 0.2404,E1 1.65,E2 202.7076} C_DIS
LIN {X -66.1413,Y -118.5408,Z 189,A -111.6568,B 1.7017,C 0.2385,E1 1.645,E2 204.7741} C_DIS
LIN {X -71.1676,Y -115.5925,Z 189,A -114.188,B 1.7021,C 0.2357,E1 1.6389,E2 207.3152} C_DIS
LIN {X -74.7062,Y -113.3375,Z 189,A -116.4472,B 1.7023,C 0.2345,E1 1.6334,E2 209.64} C_DIS
LIN {X -78.2382,Y -110.9288,Z 189,A -117.574,B 1.7028,C 0.2304,E1 1.631,E2 210.676} C_DIS
LIN {X -80.5164,Y -109.2866,Z 189,A -119.1329,B 1.7029,C 0.2296,E1 1.6274,E2 212.2851} C_DIS
LIN {X -83.883,Y -106.7242,Z 189,A -121.0231,B 1.7033,C 0.2271,E1 1.6231,E2 214.1894} C_DIS
LIN {X -87.3711,Y -103.8881,Z 189,A -123.0166,B 1.7036,C 0.2243,E1 1.6188,E2 216.1957} C_DIS
LIN {X -90.7866,Y -100.9172,Z 189,A -125.2509,B 1.704,C 0.2217,E1 1.614,E2 218.473} C_DIS
LIN {X -93.15,Y -98.739,Z 189,A -126.936,B 1.7042,C 0.22,E1 1.6105,E2 220.2016} C_DIS
LIN {X -96.4237,Y -95.5453,Z 189,A -128.5133,B 1.7047,C 0.2158,E1 1.6075,E2 221.7319} C_DIS
LIN {X -99.5966,Y -92.2338,Z 189,A -130.5686,B 1.7052,C 0.2123,E1 1.6035,E2 223.8028} C_DIS
LIN {X -102.5767,Y -88.9079,Z 189,A -132.5592,B 1.7056,C 0.2088,E1 1.5998,E2 225.8072} C_DIS
LIN {X -105.3554,Y -85.5967,Z 189,A -134.5095,B 1.706,C 0.2053,E1 1.5963,E2 227.7738} C_DIS
LIN {X -108.1081,Y -82.0927,Z 189,A -136.5433,B 1.7065,C 0.2016,E1 1.5928,E2 229.8275} C_DIS
LIN {X -110.723,Y -78.5299,Z 189,A -138.5126,B 1.7069,C 0.1978,E1 1.5896,E2 231.81} C_DIS
LIN {X -113.1677,Y -74.9642,Z 189,A -140.4484,B 1.7074,C 0.1939,E1 1.5865,E2 233.76} C_DIS
LIN {X -115.4919,Y -71.3314,Z 189,A -142.3478,B 1.7078,C 0.1898,E1 1.5837,E2 235.6693} C_DIS
LIN {X -117.6276,Y -67.7513,Z 189,A -144.2839,B 1.7082,C 0.186,E1 1.5809,E2 237.628} C_DIS
LIN {X -120.4128,Y -62.6646,Z 189,A -146.8229,B 1.7089,C 0.1802,E1 1.5775,E2 240.1781} C_DIS
LIN {X -121.8691,Y -59.7819,Z 189,A -148.3123,B 1.7092,C 0.177,E1 1.5756,E2 241.6835} C_DIS
LIN {X -123.3568,Y -56.6488,Z 189,A -149.8594,B 1.7096,C 0.1735,E1 1.5738,E2 243.2409} C_DIS
LIN {X -124.6337,Y -53.7802,Z 189,A -151.3553,B 1.7099,C 0.1704,E1 1.5721,E2 244.7585} C_DIS
LIN {X -125.9315,Y -50.6669,Z 189,A -152.8538,B 1.7102,C 0.1668,E1 1.5705,E2 246.2661} C_DIS
LIN {X -127.4885,Y -46.6149,Z 189,A -155.1116,B 1.7106,C 0.1625,E1 1.5682,E2 248.5781} C_DIS
LIN {X -129.0446,Y -42.1193,Z 189,A -157.0202,B 1.7111,C 0.1572,E1 1.5665,E2 250.4731} C_DIS
LIN {X -129.9499,Y -39.2326,Z 189,A -158.4257,B 1.7114,C 0.1539,E1 1.5654,E2 251.8946} C_DIS
LIN {X -131.1678,Y -34.9416,Z 189,A -160.5125,B 1.7119,C 0.149,E1 1.5638,E2 254.0067} C_DIS
LIN {X -132.1675,Y -30.9554,Z 189,A -162.4704,B 1.7122,C 0.1445,E1 1.5625,E2 255.9923} C_DIS
LIN {X -133.0228,Y -27.0346,Z 189,A -164.1844,B 1.7126,C 0.1399,E1 1.5615,E2 257.708} C_DIS
LIN {X -133.6565,Y -23.7053,Z 189,A -165.7696,B 1.7129,C 0.1361,E1 1.5607,E2 259.3122} C_DIS
LIN {X -134.2651,Y -19.987,Z 189,A -167.6622,B 1.7133,C 0.132,E1 1.5598,E2 261.2423} C_DIS
LIN {X -134.8051,Y -15.924,Z 189,A -169.3799,B 1.7136,C 0.1271,E1 1.5592,E2 262.9575} C_DIS
LIN {X -135.2202,Y -11.9047,Z 189,A -171.3085,B 1.714,C 0.1225,E1 1.5587,E2 264.9134} C_DIS
LIN {X -135.4946,Y -8.2003,Z 189,A -172.9495,B 1.7143,C 0.1182,E1 1.5584,E2 266.5627} C_DIS
LIN {X -135.6753,Y -4.301,Z 189,A -174.8206,B 1.7146,C 0.1137,E1 1.5582,E2 268.461} C_DIS
LIN {X -135.7441,Y -0.3548,Z 189,A -176.7381,B 1.7149,C 0.1092,E1 1.5582,E2 270.409} C_DIS
LIN {X -135.69,Y 3.7732,Z 189,A -178.4586,B 1.7152,C 0.1043,E1 1.5582,E2 272.1256} C_DIS
LIN {X -135.5533,Y 7.1719,Z 189,A 179.955,B 1.7154,C 0.1004,E1 1.5585,E2 273.7299} C_DIS
LIN {X -135.2687,Y 11.33,Z 189,A 178.0351,B 1.7157,C 0.0956,E1 1.5589,E2 275.6686} C_DIS
LIN {X -134.8966,Y 15.1419,Z 189,A 176.2277,B 1.7159,C 0.0912,E1 1.5594,E2 277.4987} C_DIS
LIN {X -134.4103,Y 18.9708,Z 189,A 174.4674,B 1.7161,C 0.0868,E1 1.56,E2 279.2741} C_DIS
LIN {X -133.8848,Y 22.3789,Z 189,A 172.9041,B 1.7163,C 0.0828,E1 1.5607,E2 280.8497} C_DIS
LIN {X -133.2686,Y 25.7979,Z 189,A 171.2929,B 1.7165,C 0.0789,E1 1.5616,E2 282.4779} C_DIS
LIN {X -132.382,Y 30.0167,Z 189,A 169.008,B 1.7167,C 0.0742,E1 1.563,E2 284.8184} C_DIS
LIN {X -131.6202,Y 33.1975,Z 189,A 168.0988,B 1.7169,C 0.0701,E1 1.5636,E2 285.6691} C_DIS
LIN {X -130.3673,Y 37.8204,Z 189,A 165.6021,B 1.7171,C 0.065,E1 1.5654,E2 288.2225} C_DIS
LIN {X -129.2421,Y 41.5022,Z 189,A 163.8929,B 1.7173,C 0.0608,E1 1.5669,E2 289.9408} C_DIS
LIN {X -128.269,Y 44.4179,Z 189,A 162.4305,B 1.7173,C 0.0575,E1 1.5682,E2 291.4224} C_DIS
LIN {X -127.0117,Y 47.8959,Z 189,A 160.7518,B 1.7175,C 0.0535,E1 1.5698,E2 293.1142} C_DIS
LIN {X -125.6259,Y 51.425,Z 189,A 158.8723,B 1.7176,C 0.0496,E1 1.5718,E2 295.0263} C_DIS
LIN {X -123.8208,Y 55.6266,Z 189,A 156.9484,B 1.7178,C 0.0447,E1 1.574,E2 296.948} C_DIS
LIN {X -122.4122,Y 58.6613,Z 189,A 155.4267,B 1.7178,C 0.0413,E1 1.5758,E2 298.4819} C_DIS
LIN {X -120.973,Y 61.5742,Z 189,A 153.8309,B 1.7179,C 0.0381,E1 1.5778,E2 300.1035} C_DIS
LIN {X -118.9388,Y 65.4227,Z 189,A 151.8502,B 1.718,C 0.0338,E1 1.5805,E2 302.1001} C_DIS
LIN {X -116.2731,Y 70.0501,Z 189,A 149.5078,B 1.718,C 0.0286,E1 1.5838,E2 304.4515} C_DIS
LIN {X -114.1207,Y 73.5053,Z 189,A 147.5887,B 1.7182,C 0.0248,E1 1.5867,E2 306.3932} C_DIS
LIN {X -111.6597,Y 77.1925,Z 189,A 145.5603,B 1.7182,C 0.0208,E1 1.5899,E2 308.4389} C_DIS
LIN {X -108.9724,Y 80.941,Z 189,A 143.4952,B 1.7182,C 0.0167,E1 1.5934,E2 310.5165} C_DIS
LIN {X -106.4161,Y 84.2742,Z 189,A 141.5653,B 1.7182,C 0.0131,E1 1.5967,E2 312.4637} C_DIS
LIN {X -102.6288,Y 88.8473,Z 189,A 138.4383,B 1.7183,C 0.0088,E1 1.6025,E2 315.6613} C_DIS
LIN {X -99.5518,Y 92.2819,Z 189,A 137.177,B 1.7183,C 0.0041,E1 1.6047,E2 316.8414} C_DIS
LIN {X -97.4764,Y 94.471,Z 189,A 135.5289,B 1.7183,C 0.0022,E1 1.608,E2 318.5325} C_DIS
LIN {X -92.7663,Y 99.1005,Z 189,A 132.2479,B 1.7183,C -0.0021,E1 1.6147,E2 321.8688} C_DIS
LIN {X -90.005,Y 101.6146,Z 189,A 131.2858,B 1.7183,C -0.0058,E1 1.6166,E2 322.7586} C_DIS
LIN {X -87.8644,Y 103.471,Z 189,A 129.6467,B 1.7183,C -0.0071,E1 1.6202,E2 324.4485} C_DIS
LIN {X -84.3427,Y 106.3615,Z 189,A 126.8368,B 1.7183,C -0.0086,E1 1.6266,E2 327.3589} C_DIS
LIN {X -79.4703,Y 110.0497,Z 189,A 124.9222,B 1.7183,C -0.0137,E1 1.6307,E2 329.1957} C_DIS
LIN {X -75.8272,Y 112.5911,Z 189,A 122.9569,B 1.7183,C -0.0161,E1 1.6353,E2 331.1703} C_DIS
LIN {X -69.0573,Y 116.8658,Z 189,A 118.8261,B 1.7183,C -0.0189,E1 1.6453,E2 335.3848} C_DIS
LIN {X -64.44,Y 119.4736,Z 189,A 117.145,B 1.7182,C -0.0227,E1 1.6493,E2 337.0011} C_DIS
LIN {X -61.4143,Y 121.0544,Z 189,A 115.7721,B 1.7182,C -0.0244,E1 1.6527,E2 338.3652} C_DIS
LIN {X -58.3803,Y 122.5464,Z 189,A 114.192,B 1.7182,C -0.0255,E1 1.6567,E2 339.9619} C_DIS
LIN {X -54.9242,Y 124.135,Z 189,A 112.6175,B 1.7182,C -0.0271,E1 1.6607,E2 341.532} C_DIS
LIN {X -52.1213,Y 125.3367,Z 189,A 111.276,B 1.7182,C -0.0281,E1 1.6642,E2 342.8788} C_DIS
LIN {X -48.7013,Y 126.7057,Z 189,A 109.7026,B 1.7181,C -0.0293,E1 1.6683,E2 344.4536} C_DIS
LIN {X -41.9635,Y 129.0947,Z 189,A 106.6711,B 1.7181,C -0.0313,E1 1.6764,E2 347.485} C_DIS
LIN {X -38.4142,Y 130.1935,Z 189,A 105.0011,B 1.7181,C -0.032,E1 1.6809,E2 349.1659} C_DIS
LIN {X -34.9793,Y 131.1578,Z 189,A 103.4538,B 1.7181,C -0.0326,E1 1.685,E2 350.717} C_DIS
LIN {X -31.7253,Y 131.9827,Z 189,A 102.0761,B 1.7181,C -0.0333,E1 1.6888,E2 352.0895} C_DIS
LIN {X -28.6165,Y 132.6915,Z 189,A 100.6848,B 1.7181,C -0.0337,E1 1.6926,E2 353.4853} C_DIS
LIN {X -25.3581,Y 133.3527,Z 189,A 99.2511,B 1.718,C -0.034,E1 1.6966,E2 354.9218} C_DIS
LIN {X -20.7714,Y 134.1436,Z 189,A 97.1185,B 1.718,C -0.034,E1 1.7025,E2 357.0726} C_DIS
LIN {X -16.5736,Y 134.7277,Z 189,A 95.4118,B 1.718,C -0.0344,E1 1.7072,E2 358.7691} C_DIS
LIN {X -12.8512,Y 135.1327,Z 189,A 93.922,B 1.718,C -0.0347,E1 1.7114,E2 360.2478} C_DIS
LIN {X -6.4253,Y 135.5908,Z 189,A 91.2237,B 1.718,C -0.0347,E1 1.7189,E2 362.9426} C_DIS
LIN {X 0.038,Y 135.7444,Z 189,A 88.5299,B 1.718,C -0.0342,E1 1.7265,E2 365.6315} C_DIS
LIN {X 3.5628,Y 135.6959,Z 189,A 86.4984,B 1.718,C -0.0317,E1 1.7323,E2 367.724} C_DIS
LIN {X 8.0237,Y 135.5055,Z 189,A 84.8464,B 1.718,C -0.0318,E1 1.7369,E2 369.349} C_DIS
LIN {X 11.3144,Y 135.2701,Z 189,A 83.8087,B 1.718,C -0.0326,E1 1.7396,E2 370.3458} C_DIS
LIN {X 14.8276,Y 134.9304,Z 189,A 82.3114,B 1.718,C -0.0318,E1 1.7438,E2 371.8434} C_DIS
LIN {X 18.7466,Y 134.4423,Z 189,A 80.3733,B 1.718,C -0.0296,E1 1.7493,E2 373.8119} C_DIS
LIN {X 21.9956,Y 133.9488,Z 189,A 79.4988,B 1.718,C -0.0308,E1 1.7516,E2 374.6274} C_DIS
LIN {X 26.7383,Y 133.0831,Z 189,A 77.2838,B 1.718,C -0.0285,E1 1.7577,E2 376.8625} C_DIS
LIN {X 30.3929,Y 132.296,Z 189,A 75.8042,B 1.7181,C -0.0277,E1 1.7617,E2 378.3304} C_DIS
LIN {X 33.4921,Y 131.5455,Z 189,A 74.4668,B 1.7181,C -0.0265,E1 1.7654,E2 379.6664} C_DIS
LIN {X 36.8742,Y 130.6381,Z 189,A 73.0514,B 1.7181,C -0.0253,E1 1.7692,E2 381.0742} C_DIS
LIN {X 40.321,Y 129.6168,Z 189,A 71.4276,B 1.7181,C -0.0233,E1 1.7736,E2 382.7099} C_DIS
LIN {X 44.4538,Y 128.2566,Z 189,A 69.1308,B 1.7182,C -0.019,E1 1.7798,E2 385.0589} C_DIS
LIN {X 49.4364,Y 126.4199,Z 189,A 67.5761,B 1.7182,C -0.0196,E1 1.7836,E2 386.5346} C_DIS
LIN {X 55.0044,Y 124.0991,Z 189,A 65.3121,B 1.7182,C -0.0177,E1 1.7894,E2 388.7656} C_DIS
LIN {X 58.9491,Y 122.2747,Z 189,A 63.4194,B 1.7182,C -0.0149,E1 1.7942,E2 390.6648} C_DIS
LIN {X 61.7901,Y 120.8631,Z 189,A 62.1464,B 1.7182,C -0.0133,E1 1.7974,E2 391.9299} C_DIS
LIN {X 64.8749,Y 119.2379,Z 189,A 59.862,B 1.7183,C -0.0068,E1 1.8032,E2 394.3079} C_DIS
LIN {X 70.4733,Y 116.0172,Z 189,A 58.394,B 1.7183,C -0.009,E1 1.8064,E2 395.6301} C_DIS
LIN {X 74.5317,Y 113.4524,Z 189,A 56.4279,B 1.7183,C -0.006,E1 1.811,E2 397.5891} C_DIS
LIN {X 76.8014,Y 111.9283,Z 189,A 54.9972,B 1.7183,C -0.0025,E1 1.8144,E2 399.0522} C_DIS
LIN {X 80.5919,Y 109.2311,Z 189,A 53.1426,B 1.7183,C 0.0004,E1 1.8186,E2 400.8941} C_DIS
LIN {X 84.0413,Y 106.5999,Z 189,A 51.4292,B 1.7183,C 0.0032,E1 1.8224,E2 402.5936} C_DIS
LIN {X 87.4816,Y 103.7953,Z 189,A 49.6344,B 1.7183,C 0.0063,E1 1.8262,E2 404.3793} C_DIS
Enddeposition()
END
